//     normal_speed_task Outputs/csp_case_main_safety_air.sis.open_output.status <-> StandardOutputs/Air.csp_case_main_safety_air.sis.open_output.status_355
//     normal_speed_task Outputs/csp_case_main_safety_drives_PS2000.sis.open_output.status <-> StandardOutputs/DrivesRackPowerSupply.csp_case_main_safety_drives_PS2000.sis.open_output.status_57
//     normal_speed_task Outputs/csp_case_main_safety_drives_SD10000.sig.safety_group_err_ack_output.status <-> StandardOutputs/SD10000.ErrorAcknowledgement_35
//     normal_speed_task Outputs/csp_case_main_safety_drives_SD10100.sig.safety_group_err_ack_output.status <-> StandardOutputs/SD10100.ErrorAcknowledgement_37
//     normal_speed_task Outputs/csp_case_main_safety_drives_SD10200.sig.safety_group_err_ack_output.status <-> StandardOutputs/SD10200.ErrorAcknowledgement_39
//     normal_speed_task Outputs/csp_case_main_safety_drives_SD10300.sig.safety_group_err_ack_output.status <-> StandardOutputs/SD10300.ErrorAcknowledgement_41
//     normal_speed_task Outputs/csp_case_main_safety_drives_SD10400.sig.safety_group_err_ack_output.status <-> StandardOutputs/SD10400.ErrorAcknowledgement_43
//     normal_speed_task Outputs/csp_case_main_safety_drives_SD11000.sig.safety_group_err_ack_output.status <-> StandardOutputs/SD11000.ErrorAcknowledgement_45
//     normal_speed_task Outputs/csp_case_main_safety_drives_SD12000.sig.safety_group_err_ack_output.status <-> StandardOutputs/SD12000.ErrorAcknowledgement_19
//     normal_speed_task Outputs/csp_case_main_safety_drives_SD15000.sig.safety_group_err_ack_output.status <-> StandardOutputs/SD15000.ErrorAcknowledgement_47
//     normal_speed_task Outputs/csp_case_main_safety_drives_SD2100.sig.safety_group_err_ack_output.status <-> StandardOutputs/SD2100.ErrorAcknowledgement_9
//     normal_speed_task Outputs/csp_case_main_safety_drives_SD2200.sig.safety_group_err_ack_output.status <-> StandardOutputs/SD2200.ErrorAcknowledgement_11
//     normal_speed_task Outputs/csp_case_main_safety_drives_SD2300.sig.safety_group_err_ack_output.status <-> StandardOutputs/SD2300.ErrorAcknowledgement_13
//     normal_speed_task Outputs/csp_case_main_safety_drives_SD2400.sig.safety_group_err_ack_output.status <-> StandardOutputs/SD2400.ErrorAcknowledgement_15
//     normal_speed_task Outputs/csp_case_main_safety_drives_SD2500.sig.safety_group_err_ack_output.status <-> StandardOutputs/SD2500.ErrorAcknowledgement_17
//     normal_speed_task Outputs/csp_case_main_safety_drives_SD26000.sig.safety_group_err_ack_output.status <-> StandardOutputs/SD26000.ErrorAcknowledgement_49
//     normal_speed_task Outputs/csp_case_main_safety_drives_SD26100.sig.safety_group_err_ack_output.status <-> StandardOutputs/SD26100.ErrorAcknowledgement_51
//     normal_speed_task Outputs/csp_case_main_safety_drives_SD8000.sig.safety_group_err_ack_output.status <-> StandardOutputs/SD8000.ErrorAcknowledgement_21
//     normal_speed_task Outputs/csp_case_main_safety_drives_SD8100.sig.safety_group_err_ack_output.status <-> StandardOutputs/SD8100.ErrorAcknowledgement_23
//     normal_speed_task Outputs/csp_case_main_safety_drives_SD8200.sig.safety_group_err_ack_output.status <-> StandardOutputs/SD8200.ErrorAcknowledgement_25
//     normal_speed_task Outputs/csp_case_main_safety_drives_SD8300.sig.safety_group_err_ack_output.status <-> StandardOutputs/SD8300.ErrorAcknowledgement_27
//     normal_speed_task Outputs/csp_case_main_safety_drives_SD8400.sig.safety_group_err_ack_output.status <-> StandardOutputs/SD8400.ErrorAcknowledgement_29
//     normal_speed_task Outputs/csp_case_main_safety_drives_SD8500.sig.safety_group_err_ack_output.status <-> StandardOutputs/SD8500.ErrorAcknowledgement_31
//     normal_speed_task Outputs/csp_case_main_safety_drives_SD8600.sig.safety_group_err_ack_output.status <-> StandardOutputs/SD8600.ErrorAcknowledgement_33
//     normal_speed_task Outputs/csp_case_main_safety_drives_SD10000.sig.safety_group_run_output.status <-> StandardOutputs/SD10000.Run_36
//     normal_speed_task Outputs/csp_case_main_safety_drives_SD10100.sig.safety_group_run_output.status <-> StandardOutputs/SD10100.Run_38
//     normal_speed_task Outputs/csp_case_main_safety_drives_SD10200.sig.safety_group_run_output.status <-> StandardOutputs/SD10200.Run_40
//     normal_speed_task Outputs/csp_case_main_safety_drives_SD10300.sig.safety_group_run_output.status <-> StandardOutputs/SD10300.Run_42
//     normal_speed_task Outputs/csp_case_main_safety_drives_SD10400.sig.safety_group_run_output.status <-> StandardOutputs/SD10400.Run_44
//     normal_speed_task Outputs/csp_case_main_safety_drives_SD11000.sig.safety_group_run_output.status <-> StandardOutputs/SD11000.Run_46
//     normal_speed_task Outputs/csp_case_main_safety_drives_SD12000.sig.safety_group_run_output.status <-> StandardOutputs/SD12000.Run_20
//     normal_speed_task Outputs/csp_case_main_safety_drives_SD15000.sig.safety_group_run_output.status <-> StandardOutputs/SD15000.Run_48
//     normal_speed_task Outputs/csp_case_main_safety_drives_SD2100.sig.safety_group_run_output.status <-> StandardOutputs/SD2100.Run_10
//     normal_speed_task Outputs/csp_case_main_safety_drives_SD2200.sig.safety_group_run_output.status <-> StandardOutputs/SD2200.Run_12
//     normal_speed_task Outputs/csp_case_main_safety_drives_SD2300.sig.safety_group_run_output.status <-> StandardOutputs/SD2300.Run_14
//     normal_speed_task Outputs/csp_case_main_safety_drives_SD2400.sig.safety_group_run_output.status <-> StandardOutputs/SD2400.Run_16
//     normal_speed_task Outputs/csp_case_main_safety_drives_SD2500.sig.safety_group_run_output.status <-> StandardOutputs/SD2500.Run_18
//     normal_speed_task Outputs/csp_case_main_safety_drives_SD26000.sig.safety_group_run_output.status <-> StandardOutputs/SD26000.Run_50
//     normal_speed_task Outputs/csp_case_main_safety_drives_SD26100.sig.safety_group_run_output.status <-> StandardOutputs/SD26100.Run_52
//     normal_speed_task Outputs/csp_case_main_safety_drives_SD8000.sig.safety_group_run_output.status <-> StandardOutputs/SD8000.Run_22
//     normal_speed_task Outputs/csp_case_main_safety_drives_SD8100.sig.safety_group_run_output.status <-> StandardOutputs/SD8100.Run_24
//     normal_speed_task Outputs/csp_case_main_safety_drives_SD8200.sig.safety_group_run_output.status <-> StandardOutputs/SD8200.Run_26
//     normal_speed_task Outputs/csp_case_main_safety_drives_SD8300.sig.safety_group_run_output.status <-> StandardOutputs/SD8300.Run_28
//     normal_speed_task Outputs/csp_case_main_safety_drives_SD8400.sig.safety_group_run_output.status <-> StandardOutputs/SD8400.Run_30
//     normal_speed_task Outputs/csp_case_main_safety_drives_SD8500.sig.safety_group_run_output.status <-> StandardOutputs/SD8500.Run_32
//     normal_speed_task Outputs/csp_case_main_safety_drives_SD8600.sig.safety_group_run_output.status <-> StandardOutputs/SD8600.Run_34
//     normal_speed_task Outputs/csp_case_main_safety_emergency.sis.open_output.status <-> StandardOutputs/EmergencyCircuit.csp_case_main_safety_emergency.sis.open_output.status_65
//     normal_speed_task Outputs/csp_case_main_safety_guards.sis.open_output.status <-> StandardOutputs/Guards.csp_case_main_safety_guards.sis.open_output.status_274
//   SFI_CasePacker Instance <-> Cabinet ethercat master/CSPENC3/SPLC5000Slot14 (EL1819)
//     highest_speed_task Inputs/csp_case_feed_arm_sensors.case_feed_pb_di.field.status <-> Channel 12/Input
//     highest_speed_task Inputs/csp_case_glue_hotMelt.feeder_faulted_di.field.status <-> Channel 4/Input
//     highest_speed_task Inputs/csp_case_glue_hotMelt.level_ok_di.field.status <-> Channel 8/Input
//     highest_speed_task Inputs/csp_case_glue_hotMelt.ready_di.field.status <-> Channel 7/Input
//     low_speed_task Inputs/csp_case_main_safety_guards.sio_door_1.protection_safely_closed_input.status <-> Channel 1/Input
//     low_speed_task Inputs/csp_case_main_safety_guards.sio_door_2.protection_safely_closed_input.status <-> Channel 2/Input
//     low_speed_task Inputs/csp_main_jogManager.di_pendant_negative.field.status <-> Channel 12/Input
//     low_speed_task Inputs/csp_main_jogManager.di_pendant_positive.field.status <-> Channel 15/Input
//     lowest_speed_task Inputs/csp_case_main_cabinet.temperature_fault_di.field.status <-> Channel 3/Input
//   SFI_CasePacker Instance <-> Cabinet ethercat master/CSPENC3/SPLC5000Slot15 (EL1819)
//     highest_speed_task Inputs/csp_transfer_infeed_barcode_reader.Good_Read <-> Channel 7/Input
//     highest_speed_task Inputs/csp_transfer_infeed_barcode_reader.No_Read <-> Channel 8/Input
//     low_speed_task Inputs/csp_case_discharge_reject_modsort.modsort_fwd_faulted_di.field.status <-> Channel 1/Input
//     low_speed_task Inputs/csp_case_discharge_reject_modsort.modsort_reject_faulted_di.field.status <-> Channel 5/Input
//     lowest_speed_task Inputs/csp_case_main_cabinet.ups_alarm_di.field.status <-> Channel 3/Input
//     lowest_speed_task Inputs/csp_case_main_cabinet.ups_battery_charge_di.field.status <-> Channel 2/Input
//     lowest_speed_task Inputs/csp_case_main_cabinet.ups_battery_mode_di.field.status <-> Channel 6/Input
//   SFI_CasePacker Instance <-> Cabinet ethercat master/CSPENC3/SPLC5000Slot16 (EL2008)
//     highest_speed_task Outputs/csp_case_glue_hotMelt.standby_do.field.status <-> Channel 2/Output
//     normal_speed_task Outputs/csp_case_main_services.lights_on_do.field.status <-> Channel 8/Output
//     normal_speed_task Outputs/csp_case_main_services_airPressure.air_enable.field.status <-> Channel 7/Output
//     normal_speed_task Outputs/csp_case_main_services_pushbuttons.emergency_close_lamp_do.field.status <-> Channel 1/Output
//   SFI_CasePacker Instance <-> Cabinet ethercat master/CSPENC3/SPLC5000Slot17 (EL2008)
//     highest_speed_task Outputs/csp_case_discharge_reject_modsort.MODSORT_FWD_RUN_do.field.status <-> Channel 1/Output
//     highest_speed_task Outputs/csp_transfer_infeed_barcode_reader.Read_trigger <-> Channel 8/Output
//     highest_speed_task Outputs/csp_transfer_infeed_barcode_reader.teach_code_active <-> Channel 7/Output
//     normal_speed_task Outputs/csp_case_discharge_reject_modsort.MODSORT_REJECT_RUN_do.field.status <-> Channel 2/Output
//   SFI_CasePacker Instance <-> Cabinet ethercat master/CSPENC3/SPLC5000Slot18 (EL2008)
//     highest_speed_task Outputs/csp_transfer_infeed.temp_belt_run <-> Channel 1/Output
//   SFI_CasePacker Instance <-> Cabinet ethercat master/CSPENC3/SPLC5000Slot19 (EL6224)
//     highest_speed_task Inputs/csp_case_feed_arm_sensors.rfid_input_buffer.ByteArr[0] <-> IO-Link Port3_in/Bitheader 1
//     highest_speed_task Inputs/csp_case_feed_arm_sensors.rfid_input_buffer.ByteArr[9] <-> IO-Link Port3_in/Bitheader 2
//     highest_speed_task Inputs/csp_case_feed_arm_sensors.rfid_input_buffer.ByteArr[{1..8}] <-> IO-Link Port3_in/Byte {1..8}  (8 links)
//     highest_speed_task Inputs/csp_main_services.pressure_switch_value <-> IO-Link Port2/Pressure
//     highest_speed_task Outputs/csp_case_feed_arm_sensors.rfid_output_buffer.ByteArr[0] <-> IO-Link Port3_out/Bitheader 1
//     highest_speed_task Outputs/csp_case_feed_arm_sensors.rfid_output_buffer.ByteArr[9] <-> IO-Link Port3_out/Bitheader 2
//     highest_speed_task Outputs/csp_case_feed_arm_sensors.rfid_output_buffer.ByteArr[{1..8}] <-> IO-Link Port3_out/Byte {1..8}  (8 links)
//     normal_speed_task Inputs/csp_main_services.iol_master_el6224_IO6100.CONVERSION_private.process_data_input.AoeNetId <-> InfoData/AoeNetId
//     normal_speed_task Inputs/csp_main_services.iol_master_el6224_IO6100.CONVERSION_private.process_data_input.IOLinkDeviceStateInputs <-> DeviceState Inputs/State Ch1
//     normal_speed_task Inputs/csp_main_services.iol_master_el6224_IO6100.CONVERSION_private.process_data_input.IOLinkDeviceStateInputs @bit 8 <-> DeviceState Inputs/State Ch2
//     normal_speed_task Inputs/csp_main_services.iol_master_el6224_IO6100.CONVERSION_private.process_data_input.IOLinkDeviceStateInputs @bit 16 <-> DeviceState Inputs/State Ch3
//     normal_speed_task Inputs/csp_main_services.iol_master_el6224_IO6100.CONVERSION_private.process_data_input.IOLinkDeviceStateInputs @bit 24 <-> DeviceState Inputs/State Ch4
//     normal_speed_task Outputs/csp_main_services_towerLamp.buzzer_do.field.status <-> IO-Link Port1_out/Buzzer State
//     normal_speed_task Outputs/csp_main_services_towerLamp.buzzer_volume <-> IO-Link Port1_out/Buzzer Volume
//     normal_speed_task Outputs/csp_main_services_towerLamp.tower_lamp.iol_slave_pdo_output.blinking_freq <-> IO-Link Port1_out/Blinking frequency / Level value high byte / Running speed
//     normal_speed_task Outputs/csp_main_services_towerLamp.tower_lamp.iol_slave_pdo_output.number_segments <-> IO-Link Port1_out/Number of segments / Level type
//     normal_speed_task Outputs/csp_main_services_towerLamp.tower_lamp.iol_slave_pdo_output.operating_mode <-> IO-Link Port1_out/Operating mode
//     normal_speed_task Outputs/csp_main_services_towerLamp.tower_lamp.iol_slave_pdo_output.seg_1_blink <-> IO-Link Port1_out/Segment 1 blink / dominant / LED4
//     normal_speed_task Outputs/csp_main_services_towerLamp.tower_lamp.iol_slave_pdo_output.seg_2_blink <-> IO-Link Port1_out/Segment 2 blink / dominant / LED8
//     normal_speed_task Outputs/csp_main_services_towerLamp.tower_lamp.iol_slave_pdo_output.seg_3_blink <-> IO-Link Port1_out/Segment 3 blink / dominant / LED12
//     normal_speed_task Outputs/csp_main_services_towerLamp.tower_lamp.iol_slave_pdo_output.seg_1_color <-> IO-Link Port1_out/Segment 1 color / Background color / LED3-1
//     normal_speed_task Outputs/csp_main_services_towerLamp.tower_lamp.iol_slave_pdo_output.seg_2_color <-> IO-Link Port1_out/Segment 2 color / Running color / LED7-5
//     normal_speed_task Outputs/csp_main_services_towerLamp.tower_lamp.iol_slave_pdo_output.seg_3_color <-> IO-Link Port1_out/Segment 3 color / LED11-9
//   SFI_CasePacker Instance <-> Cabinet ethercat master/CSPENC3/SPLC5000Slot20 (EL4004)
//     normal_speed_task Outputs/csp_case_discharge_reject.modsort_belt_speed_analog_reference_ao.field.value <-> AO Outputs Channel 1/Analog output
//   SFI_CasePacker Instance <-> Cabinet ethercat master/CSPENC3/SPLC5000Slot21(EK1122-0008)/Box 92 (EP2328-0001)
//     highest_speed_task Outputs/csp_case_glue.os_lower_gun_1_do.field.status <-> Channel 7/Output
//     highest_speed_task Outputs/csp_case_glue.os_lower_gun_2_do.field.status <-> Channel 8/Output
//     highest_speed_task Outputs/csp_case_glue.os_upper_gun_1_do.field.status <-> Channel 5/Output
//     highest_speed_task Outputs/csp_case_glue.os_upper_gun_2_do.field.status <-> Channel 6/Output
//   SFI_CasePacker Instance <-> Cabinet ethercat master/CSPENC3/SPLC5000Slot21(EK1122-0008)/Box 93 (EP2328-0001)
//     highest_speed_task Outputs/csp_case_glue.ls_lower_gun_1_do.field.status <-> Channel 7/Output
//     highest_speed_task Outputs/csp_case_glue.ls_lower_gun_2_do.field.status <-> Channel 8/Output
//     highest_speed_task Outputs/csp_case_glue.ls_upper_gun_1_do.field.status <-> Channel 5/Output
//     highest_speed_task Outputs/csp_case_glue.ls_upper_gun_2_do.field.status <-> Channel 6/Output
//   SFI_CasePacker Instance <-> Cabinet ethercat master/CSPENC3/SPLC5000Slot21(EK1122-0008)/IOB11120 (EP1018-0001)
//     highest_speed_task Inputs/csp_case_fc_ls_upper_sensors.flap_di.field.status <-> Channel 3/Input
//     highest_speed_task Inputs/csp_case_glue_sensors.case_present_ls_di.field.status <-> Channel 4/Input
//     normal_speed_task Inputs/csp_case_openFlap_sensors.open_flap_ls_di.field.status <-> Channel 2/Input
//   SFI_CasePacker Instance <-> Cabinet ethercat master/CSPENC3/SPLC5000Slot21(EK1122-0008)/IOB11130 (EP1018-0001)
//     highest_speed_task Inputs/csp_case_fc_os_upper_sensors.flap_di.field.status <-> Channel 3/Input
//     highest_speed_task Inputs/csp_case_glue_sensors.case_present_os_di.field.status <-> Channel 4/Input
//     normal_speed_task Inputs/csp_case_openFlap_sensors.open_flap_os_di.field.status <-> Channel 2/Input
//   SFI_CasePacker Instance <-> Cabinet ethercat master/CSPENC3/SPLC5000Slot21(EK1122-0008)/IOB15120 (EP1018-0001)
//     low_speed_task Inputs/csp_case_discharge_reject_sensors.downstream_backup_di.field.status <-> Channel 2/Input
//     low_speed_task Inputs/csp_case_discharge_reject_sensors.reject_backup_di.field.status <-> Channel 3/Input
//     low_speed_task Inputs/csp_case_discharge_reject_sensors.reject_present_di.field.status <-> Channel 4/Input
//     normal_speed_task Inputs/csp_case_discharge_reject_sensors.reject_trigger_di.field.status <-> Channel 1/Input
//   SFI_CasePacker Instance <-> Cabinet ethercat master/CSPENC3/SPLC5000Slot21(EK1122-0008)/IOB8800 (EP2318-0001)
//     highest_speed_task Inputs/csp_case_feed_arm_sensors.case_check_di.field.status <-> Channel 1/Input
//     highest_speed_task Outputs/csp_case_feed_arm_sensors.major_vacuum_do.field.status <-> Channel 5/Output
//     highest_speed_task Outputs/csp_case_feed_arm_sensors.minor_vacuum_do.field.status <-> Channel 7/Output
//     low_speed_task Outputs/csp_case_tr_accU_virtualMaster.brake_release_do.field.status <-> Channel 6/Output
//   SFI_CasePacker Instance <-> Cabinet ethercat master/HMI6600 (CPXXXX-BK1150)
//     normal_speed_task Inputs/csp_case_main_services_pushbuttons.reset_di.field.status <-> Term 2 (CPx9xx-8)/Channel 1/Key 1
//     normal_speed_task Inputs/csp_case_main_services_pushbuttons.start_di.field.status <-> Term 2 (CPx9xx-8)/Channel 1/Key 3
//     normal_speed_task Inputs/csp_case_main_services_pushbuttons.stop_di.field.status <-> Term 2 (CPx9xx-8)/Channel 1/Key 2
//     normal_speed_task Outputs/csp_case_main_services_pushbuttons.reset_lamp_do.field.status <-> Term 2 (CPx9xx-8)/Channel 1/LED 1
//     normal_speed_task Outputs/csp_case_main_services_pushbuttons.start_lamp_do.field.status <-> Term 2 (CPx9xx-8)/Channel 1/LED 3
//     normal_speed_task Outputs/csp_case_main_services_pushbuttons.stop_lamp_do.field.status <-> Term 2 (CPx9xx-8)/Channel 1/LED 2
//   SFI_CasePacker Instance <-> Cabinet ethercat master/IO61000 (EK1100)/IO6100Slot24 (EL7211)
//     low_speed_task Inputs/csp_case_transport_accU_depth.Slot24_drv.process_data_input.status_word <-> DRV Statusword/Statusword
//     low_speed_task Inputs/csp_case_transport_accU_depth.axis.hard_increments.value <-> FB Position/Position
//     lowest_speed_task Inputs/csp_case_transport_accU_depth.NC_encoder_val <-> FB Position/Position
//   SFI_CasePacker Instance <-> Cabinet ethercat master/IO61000 (EK1100)/IO6100Slot26 (EL7211)
//     low_speed_task Inputs/csp_case_feed_shuttle_accU_depth.Slot26_drv.process_data_input.status_word <-> DRV Statusword/Statusword
//     low_speed_task Inputs/csp_case_feed_shuttle_accU_depth.axis.hard_increments.value <-> FB Position/Position
//     lowest_speed_task Inputs/csp_case_feed_shuttle_accU_depth.NC_encoder_val <-> FB Position/Position
//   SFI_CasePacker Instance <-> Cabinet ethercat master/IO61000 (EK1100)/IO6100Slot29 (EL7211)
//     low_speed_task Inputs/csp_case_feed_magazine_accU_lsDepth.Slot29_drv.process_data_input.status_word <-> DRV Statusword/Statusword
//     low_speed_task Inputs/csp_case_feed_magazine_accU_lsDepth.axis.hard_increments.value <-> FB Position/Position
//     lowest_speed_task Inputs/csp_case_feed_magazine_accU_lsDepth.NC_encoder_val <-> FB Position/Position
//   SFI_CasePacker Instance <-> Cabinet ethercat master/IO61000 (EK1100)/IO6100Slot31 (EL7211)
//     low_speed_task Inputs/csp_case_feed_magazine_accU_osDepth.Slot31_drv.process_data_input.status_word <-> DRV Statusword/Statusword
//     low_speed_task Inputs/csp_case_feed_magazine_accU_osDepth.axis.hard_increments.value <-> FB Position/Position
//     lowest_speed_task Inputs/csp_case_feed_magazine_accU_osDepth.NC_encoder_val <-> FB Position/Position
//   SFI_CasePacker Instance <-> Cabinet ethercat master/IO61000 (EK1100)/IO6100Slot34 (EL7221)
//     low_speed_task Inputs/csp_case_loader_guide_accU_width.Slot34_drv.process_data_input.status_word <-> DRV Statusword/Statusword
//     low_speed_task Inputs/csp_case_loader_guide_accU_width.axis.hard_increments.value <-> FB Position/Position
//     lowest_speed_task Inputs/csp_case_loader_guide_accU_width.NC_encoder_val <-> FB Position/Position
//   SFI_CasePacker Instance <-> Cabinet ethercat master/IO61000 (EK1100)/IO6100Slot36 (EL7211)
//     low_speed_task Inputs/csp_case_glue_os_accU_width.Slot36_drv.process_data_input.status_word <-> DRV Statusword/Statusword
//     low_speed_task Inputs/csp_case_glue_os_accU_width.axis.hard_increments.value <-> FB Position/Position
//     lowest_speed_task Inputs/csp_case_glue_os_accU_width.NC_encoder_val <-> FB Position/Position
//   SFI_CasePacker Instance <-> Cabinet ethercat master/IO61000 (EK1100)/IO6100Slot39 (EL7211)
//     low_speed_task Inputs/csp_case_glue_os_accU_upperPosition.Slot39_drv.process_data_input.status_word <-> DRV Statusword/Statusword
//     low_speed_task Inputs/csp_case_glue_os_accU_upperPosition.axis.hard_increments.value <-> FB Position/Position
//     lowest_speed_task Inputs/csp_case_glue_os_accU_upperPosition.NC_encoder_val <-> FB Position/Position
//   SFI_CasePacker Instance <-> Cabinet ethercat master/IO61000 (EK1100)/IO6100Slot41 (EL7211)
//     low_speed_task Inputs/csp_case_glue_os_accU_lowerPosition.Slot41_drv.process_data_input.status_word <-> DRV Statusword/Statusword
//     low_speed_task Inputs/csp_case_glue_os_accU_lowerPosition.axis.hard_increments.value <-> FB Position/Position
//     lowest_speed_task Inputs/csp_case_glue_os_accU_lowerPosition.NC_encoder_val <-> FB Position/Position
//   SFI_CasePacker Instance <-> Cabinet ethercat master/IO61000 (EK1100)/IO6100Slot44 (EL7211)
//     low_speed_task Inputs/csp_case_glue_ls_accU_upperPosition.Slot44_drv.process_data_input.status_word <-> DRV Statusword/Statusword
//     low_speed_task Inputs/csp_case_glue_ls_accU_upperPosition.axis.hard_increments.value <-> FB Position/Position
//     lowest_speed_task Inputs/csp_case_glue_ls_accU_upperPosition.NC_encoder_val <-> FB Position/Position
//   SFI_CasePacker Instance <-> Cabinet ethercat master/IO61000 (EK1100)/IO6100Slot46 (EL7211)
//     low_speed_task Inputs/csp_case_glue_ls_accU_lowerPosition.Slot46_drv.process_data_input.status_word <-> DRV Statusword/Statusword
//     low_speed_task Inputs/csp_case_glue_ls_accU_lowerPosition.axis.hard_increments.value <-> FB Position/Position
//     lowest_speed_task Inputs/csp_case_glue_ls_accU_lowerPosition.NC_encoder_val <-> FB Position/Position
//   SFI_CasePacker Instance <-> Cabinet ethercat master/IO61000 (EK1100)/IO6100Slot49 (EL7211)
//     low_speed_task Inputs/csp_case_feed_reject_accU_depth.Slot49_drv.process_data_input.status_word <-> DRV Statusword/Statusword
//     low_speed_task Inputs/csp_case_feed_reject_accU_depth.axis.hard_increments.value <-> FB Position/Position
//     lowest_speed_task Inputs/csp_case_feed_reject_accU_depth.NC_encoder_val <-> FB Position/Position
//   SFI_CasePacker Instance <-> Cabinet ethercat master/IO61000 (EK1100)/IO6100Slot51 (EL7211)
//     low_speed_task Inputs/csp_case_tr_accU_os_width.Slot51_drv.process_data_input.status_word <-> DRV Statusword/Statusword
//     low_speed_task Inputs/csp_case_tr_accU_os_width.axis.hard_increments.value <-> FB Position/Position
//     lowest_speed_task Inputs/csp_case_tr_accU_os_width.NC_encoder_val <-> FB Position/Position
//   SFI_CasePacker Instance <-> Cabinet ethercat master/IO61000 (EK1100)/IO6100Slot55 (EL7211)
//     low_speed_task Inputs/csp_case_tr_accU_ls_width.Slot55_drv.process_data_input.status_word <-> DRV Statusword/Statusword
//     low_speed_task Inputs/csp_case_tr_accU_ls_width.axis.hard_increments.value <-> FB Position/Position
//     lowest_speed_task Inputs/csp_case_tr_accU_ls_width.NC_encoder_val <-> FB Position/Position
//   SFI_CasePacker Instance <-> Cabinet ethercat master/IO61000 (EK1100)/IO6100Slot57 (EL7211)
//     low_speed_task Inputs/csp_case_tr_accU_depth.Slot57_drv.process_data_input.status_word <-> DRV Statusword/Statusword
//     low_speed_task Inputs/csp_case_tr_accU_depth.axis.hard_increments.value <-> FB Position/Position
//     lowest_speed_task Inputs/csp_case_tr_accU_depth.NC_encoder_val <-> FB Position/Position
//   SFI_CasePacker Instance <-> Cabinet ethercat master/IOB2820 (EP2318-0001)
//     highest_speed_task Inputs/csp_case_fc_ls_lower_sensors.flap_di.field.status <-> Channel 1/Input
//     normal_speed_task Inputs/csp_case_openFlap_sensors.open_trailing_minor_di.field.status <-> Channel 3/Input
//   SFI_CasePacker Instance <-> Cabinet ethercat master/IOB2830 (EP2318-0001)
//     highest_speed_task Inputs/csp_case_fc_os_lower_sensors.flap_di.field.status <-> Channel 2/Input
//     low_speed_task Inputs/csp_case_transport_os_minorPlow.bwd_di.field.status <-> Channel 4/Input
//     low_speed_task Inputs/csp_case_transport_os_minorPlow.fwd_di.field.status <-> Channel 3/Input
//     normal_speed_task Inputs/csp_case_flapControl_backStop.present_di.field.status <-> Channel 1/Input
//     normal_speed_task Outputs/csp_case_flapControl_backStop.extend_do.field.status <-> Channel 5/Output
//     normal_speed_task Outputs/csp_case_transport_tensioner.chain_tensioner_do.field.status <-> Channel 7/Output
//   SFI_CasePacker Instance <-> Cabinet ethercat master/IOB3020 (EP6224-2022)
//     highest_speed_task Inputs/csp_case_closing.ls_rfid_input_buffer.ByteArr[0] <-> IO-Link Port3_in/Bitheader 1
//     highest_speed_task Inputs/csp_case_closing.ls_rfid_input_buffer.ByteArr[9] <-> IO-Link Port3_in/Bitheader 2
//     highest_speed_task Inputs/csp_case_closing.ls_rfid_input_buffer.ByteArr[{1..8}] <-> IO-Link Port3_in/Byte {1..8}  (8 links)
//     highest_speed_task Outputs/csp_case_closing.ls_rfid_output_buffer.ByteArr[0] <-> IO-Link Port3_out/Bitheader 1
//     highest_speed_task Outputs/csp_case_closing.ls_rfid_output_buffer.ByteArr[9] <-> IO-Link Port3_out/Bitheader 2
//     highest_speed_task Outputs/csp_case_closing.ls_rfid_output_buffer.ByteArr[{1..8}] <-> IO-Link Port3_out/Byte {1..8}  (8 links)
//     normal_speed_task Inputs/csp_case_loader_sensors.rfid_input_buffer.ByteArr[0] <-> IO-Link Port2_in/Bitheader 1
//     normal_speed_task Inputs/csp_case_loader_sensors.rfid_input_buffer.ByteArr[9] <-> IO-Link Port2_in/Bitheader 2
//     normal_speed_task Inputs/csp_case_loader_sensors.rfid_input_buffer.ByteArr[{1..8}] <-> IO-Link Port2_in/Byte {1..8}  (8 links)
//     normal_speed_task Outputs/csp_case_loader_sensors.rfid_output_buffer.ByteArr[0] <-> IO-Link Port2_out/Bitheader 1
//     normal_speed_task Outputs/csp_case_loader_sensors.rfid_output_buffer.ByteArr[9] <-> IO-Link Port2_out/Bitheader 2
//     normal_speed_task Outputs/csp_case_loader_sensors.rfid_output_buffer.ByteArr[{1..8}] <-> IO-Link Port2_out/Byte {1..8}  (8 links)
//   SFI_CasePacker Instance <-> Cabinet ethercat master/IOB3030 (EP6224-2022)
//     highest_speed_task Inputs/csp_case_closing.os_rfid_input_buffer.ByteArr[0] <-> IO-Link Port3_in/Bitheader 1
//     highest_speed_task Inputs/csp_case_closing.os_rfid_input_buffer.ByteArr[9] <-> IO-Link Port3_in/Bitheader 2
//     highest_speed_task Inputs/csp_case_closing.os_rfid_input_buffer.ByteArr[{1..8}] <-> IO-Link Port3_in/Byte {1..8}  (8 links)
//     highest_speed_task Outputs/csp_case_closing.os_rfid_output_buffer.ByteArr[0] <-> IO-Link Port3_out/Bitheader 1
//     highest_speed_task Outputs/csp_case_closing.os_rfid_output_buffer.ByteArr[9] <-> IO-Link Port3_out/Bitheader 2
//     highest_speed_task Outputs/csp_case_closing.os_rfid_output_buffer.ByteArr[{1..8}] <-> IO-Link Port3_out/Byte {1..8}  (8 links)
//   SFI_CasePacker Instance <-> Cabinet ethercat master/IOB8810 (EP2008-0001)
//     low_speed_task Outputs/csp_case_feed_magazine_ls_pusher.retract_do.field.status <-> Channel 2/Output
//     low_speed_task Outputs/csp_case_feed_magazine_ls_pusherTilt.extend_do.field.status <-> Channel 4/Output
//     low_speed_task Outputs/csp_case_feed_magazine_os_pusher.retract_do.field.status <-> Channel 1/Output
//     low_speed_task Outputs/csp_case_feed_magazine_os_pusherTilt.extend_do.field.status <-> Channel 3/Output
//   SFI_CasePacker Instance <-> Cabinet ethercat master/IOB8820 (EP1018-0001)
//     low_speed_task Inputs/csp_case_feed_magazine_level_zone4.di.field.status <-> Channel 1/Input
//     normal_speed_task Inputs/csp_case_feed_magazine_level_zone2.di.field.status <-> Channel 3/Input
//     normal_speed_task Inputs/csp_case_feed_magazine_level_zone3.di.field.status <-> Channel 2/Input
//     normal_speed_task Inputs/csp_case_feed_magazine_ls_pusher.retracted_di.field.status <-> Channel 6/Input
//     normal_speed_task Inputs/csp_case_feed_magazine_ls_pusherTilt.upstream_di.field.status <-> Channel 7/Input
//   SFI_CasePacker Instance <-> Cabinet ethercat master/IOB8830 (EP1018-0001)
//     low_speed_task Inputs/csp_case_feed_magazine_ls_pusherTilt.downstream_di.field.status <-> Channel 6/Input
//     low_speed_task Inputs/csp_case_feed_magazine_ls_sensors.feed_di.field.status <-> Channel 2/Input
//     normal_speed_task Inputs/csp_case_feed_magazine_level_zone1.di.field.status <-> Channel 4/Input
//     normal_speed_task Inputs/csp_case_feed_magazine_level_zonelow.di.field.status <-> Channel 5/Input
//     normal_speed_task Inputs/csp_case_feed_magazine_level_zonemin.di.field.status <-> Channel 3/Input
//   SFI_CasePacker Instance <-> Cabinet ethercat master/IOB8900 (EP1018-0001)
//     low_speed_task Inputs/csp_case_feed_magazine_os_pusherTilt.downstream_di.field.status <-> Channel 4/Input
//     low_speed_task Inputs/csp_case_feed_magazine_os_sensors.feed_di.field.status <-> Channel 3/Input
//     normal_speed_task Inputs/csp_case_feed_magazine_os_pusher.retracted_di.field.status <-> Channel 1/Input
//     normal_speed_task Inputs/csp_case_feed_magazine_os_pusherTilt.upstream_di.field.status <-> Channel 2/Input
//   SFI_CasePacker Instance <-> Cabinet ethercat master/MAN8920 (CPX-FB37)
//     highest_speed_task Outputs/csp_case_feed_shuttle_sensors.vacuum1_do.field.status <-> Module 3 (VTSA DIL 4 [32DO])/Outputs/Output 0
//     highest_speed_task Outputs/csp_case_feed_shuttle_sensors.vacuum2_do.field.status <-> Module 3 (VTSA DIL 4 [32DO])/Outputs/Output 1
//     highest_speed_task Outputs/csp_case_feed_shuttle_sensors.vacuum3_do.field.status <-> Module 3 (VTSA DIL 4 [32DO])/Outputs/Output 3
//     highest_speed_task Outputs/csp_case_feed_shuttle_sensors.vacuum4_do.field.status <-> Module 3 (VTSA DIL 4 [32DO])/Outputs/Output 2
//     highest_speed_task Outputs/csp_case_feed_shuttle_sensors.vacuum5_do.field.status <-> Module 3 (VTSA DIL 4 [32DO])/Outputs/Output 4
//     highest_speed_task Outputs/csp_case_feed_shuttle_sensors.vacuum6_do.field.status <-> Module 3 (VTSA DIL 4 [32DO])/Outputs/Output 5
//     highest_speed_task Outputs/csp_case_feed_shuttle_sensors.vacuum7_do.field.status <-> Module 3 (VTSA DIL 4 [32DO])/Outputs/Output 6
//   SFI_CasePacker Instance <-> Cabinet ethercat master/SD10000
//     highest_speed_task Inputs/csp_case_main_drives.SD10000_drv.channel_a.process_data_input.dc_bus_power <-> AT 1/DC bus power
//     highest_speed_task Inputs/csp_case_main_drives.SD10000_drv.channel_a.process_data_input.dc_bus_voltage <-> AT 1/DC bus voltage
//     highest_speed_task Inputs/csp_case_main_drives.SD10000_drv.channel_a.process_data_input.motor_temperature <-> AT 1/Motor temperature
//     highest_speed_task Inputs/csp_case_main_drives.SD10000_drv.channel_b.process_data_input.dc_bus_power <-> AT 2/DC bus power
//     highest_speed_task Inputs/csp_case_main_drives.SD10000_drv.channel_b.process_data_input.dc_bus_voltage <-> AT 2/DC bus voltage
//     highest_speed_task Inputs/csp_case_main_drives.SD10000_drv.channel_b.process_data_input.motor_temperature <-> AT 2/Motor temperature
//     normal_speed_task Inputs/csp_case_main_drives.SD10000_drv.channel_a.process_data_input.actual_absolute_current <-> AT 1/Torque-generating current, actual value
//     normal_speed_task Inputs/csp_case_main_drives.SD10000_drv.channel_a.process_data_input.dc_bus_ready <-> AT 1/Device control: Status word[15]
//     normal_speed_task Inputs/csp_case_main_drives.SD10000_drv.channel_a.process_data_input.status_parametrization_level <-> AT 1/Status parametrization level
//     normal_speed_task Inputs/csp_case_main_drives.SD10000_drv.channel_a.process_data_input.warning_active <-> AT 1/Device control: Status word[2]
//     normal_speed_task Inputs/csp_case_main_drives.SD10000_drv.channel_b.process_data_input.actual_absolute_current <-> AT 2/Torque-generating current, actual value
//     normal_speed_task Inputs/csp_case_main_drives.SD10000_drv.channel_b.process_data_input.dc_bus_ready <-> AT 2/Device control: Status word[15]
//     normal_speed_task Inputs/csp_case_main_drives.SD10000_drv.channel_b.process_data_input.status_parametrization_level <-> AT 2/Status parametrization level
//     normal_speed_task Inputs/csp_case_main_drives.SD10000_drv.channel_b.process_data_input.warning_active <-> AT 2/Device control: Status word[2]
//   SFI_CasePacker Instance <-> Cabinet ethercat master/SD10100
//     highest_speed_task Inputs/csp_case_main_drives.SD10100_drv.channel_a.process_data_input.dc_bus_power <-> AT 1/DC bus power
//     highest_speed_task Inputs/csp_case_main_drives.SD10100_drv.channel_a.process_data_input.dc_bus_voltage <-> AT 1/DC bus voltage
//     highest_speed_task Inputs/csp_case_main_drives.SD10100_drv.channel_a.process_data_input.motor_temperature <-> AT 1/Motor temperature
//     highest_speed_task Inputs/csp_case_main_drives.SD10100_drv.channel_b.process_data_input.dc_bus_power <-> AT 2/DC bus power
//     highest_speed_task Inputs/csp_case_main_drives.SD10100_drv.channel_b.process_data_input.dc_bus_voltage <-> AT 2/DC bus voltage
//     highest_speed_task Inputs/csp_case_main_drives.SD10100_drv.channel_b.process_data_input.motor_temperature <-> AT 2/Motor temperature
//     normal_speed_task Inputs/csp_case_main_drives.SD10100_drv.channel_a.process_data_input.actual_absolute_current <-> AT 1/Torque-generating current, actual value
//     normal_speed_task Inputs/csp_case_main_drives.SD10100_drv.channel_a.process_data_input.dc_bus_ready <-> AT 1/Device control: Status word[15]
//     normal_speed_task Inputs/csp_case_main_drives.SD10100_drv.channel_a.process_data_input.status_parametrization_level <-> AT 1/Status parametrization level
//     normal_speed_task Inputs/csp_case_main_drives.SD10100_drv.channel_a.process_data_input.warning_active <-> AT 1/Device control: Status word[2]
//     normal_speed_task Inputs/csp_case_main_drives.SD10100_drv.channel_b.process_data_input.actual_absolute_current <-> AT 2/Torque-generating current, actual value
//     normal_speed_task Inputs/csp_case_main_drives.SD10100_drv.channel_b.process_data_input.dc_bus_ready <-> AT 2/Device control: Status word[15]
//     normal_speed_task Inputs/csp_case_main_drives.SD10100_drv.channel_b.process_data_input.status_parametrization_level <-> AT 2/Status parametrization level
//     normal_speed_task Inputs/csp_case_main_drives.SD10100_drv.channel_b.process_data_input.warning_active <-> AT 2/Device control: Status word[2]
//   SFI_CasePacker Instance <-> Cabinet ethercat master/SD10200
//     highest_speed_task Inputs/csp_case_main_drives.SD10200_drv.channel_a.process_data_input.dc_bus_power <-> AT 1/DC bus power
//     highest_speed_task Inputs/csp_case_main_drives.SD10200_drv.channel_a.process_data_input.dc_bus_voltage <-> AT 1/DC bus voltage
//     highest_speed_task Inputs/csp_case_main_drives.SD10200_drv.channel_a.process_data_input.motor_temperature <-> AT 1/Motor temperature
//     highest_speed_task Inputs/csp_case_main_drives.SD10200_drv.channel_b.process_data_input.dc_bus_power <-> AT 2/DC bus power
//     highest_speed_task Inputs/csp_case_main_drives.SD10200_drv.channel_b.process_data_input.dc_bus_voltage <-> AT 2/DC bus voltage
//     highest_speed_task Inputs/csp_case_main_drives.SD10200_drv.channel_b.process_data_input.motor_temperature <-> AT 2/Motor temperature
//     normal_speed_task Inputs/csp_case_main_drives.SD10200_drv.channel_a.process_data_input.actual_absolute_current <-> AT 1/Torque-generating current, actual value
//     normal_speed_task Inputs/csp_case_main_drives.SD10200_drv.channel_a.process_data_input.dc_bus_ready <-> AT 1/Device control: Status word[15]
//     normal_speed_task Inputs/csp_case_main_drives.SD10200_drv.channel_a.process_data_input.status_parametrization_level <-> AT 1/Status parametrization level
//     normal_speed_task Inputs/csp_case_main_drives.SD10200_drv.channel_a.process_data_input.warning_active <-> AT 1/Device control: Status word[2]
//     normal_speed_task Inputs/csp_case_main_drives.SD10200_drv.channel_b.process_data_input.actual_absolute_current <-> AT 2/Torque-generating current, actual value
//     normal_speed_task Inputs/csp_case_main_drives.SD10200_drv.channel_b.process_data_input.dc_bus_ready <-> AT 2/Device control: Status word[15]
//     normal_speed_task Inputs/csp_case_main_drives.SD10200_drv.channel_b.process_data_input.status_parametrization_level <-> AT 2/Status parametrization level
//     normal_speed_task Inputs/csp_case_main_drives.SD10200_drv.channel_b.process_data_input.warning_active <-> AT 2/Device control: Status word[2]
//   SFI_CasePacker Instance <-> Cabinet ethercat master/SD10300
//     highest_speed_task Inputs/csp_case_main_drives.SD10300_drv.channel_a.process_data_input.dc_bus_power <-> AT 1/DC bus power
//     highest_speed_task Inputs/csp_case_main_drives.SD10300_drv.channel_a.process_data_input.dc_bus_voltage <-> AT 1/DC bus voltage
//     highest_speed_task Inputs/csp_case_main_drives.SD10300_drv.channel_a.process_data_input.motor_temperature <-> AT 1/Motor temperature
//     highest_speed_task Inputs/csp_case_main_drives.SD10300_drv.channel_b.process_data_input.dc_bus_power <-> AT 2/DC bus power
//     highest_speed_task Inputs/csp_case_main_drives.SD10300_drv.channel_b.process_data_input.dc_bus_voltage <-> AT 2/DC bus voltage
//     highest_speed_task Inputs/csp_case_main_drives.SD10300_drv.channel_b.process_data_input.motor_temperature <-> AT 2/Motor temperature
//     normal_speed_task Inputs/csp_case_main_drives.SD10300_drv.channel_a.process_data_input.actual_absolute_current <-> AT 1/Torque-generating current, actual value
//     normal_speed_task Inputs/csp_case_main_drives.SD10300_drv.channel_a.process_data_input.dc_bus_ready <-> AT 1/Device control: Status word[15]
//     normal_speed_task Inputs/csp_case_main_drives.SD10300_drv.channel_a.process_data_input.status_parametrization_level <-> AT 1/Status parametrization level
//     normal_speed_task Inputs/csp_case_main_drives.SD10300_drv.channel_a.process_data_input.warning_active <-> AT 1/Device control: Status word[2]
//     normal_speed_task Inputs/csp_case_main_drives.SD10300_drv.channel_b.process_data_input.actual_absolute_current <-> AT 2/Torque-generating current, actual value
//     normal_speed_task Inputs/csp_case_main_drives.SD10300_drv.channel_b.process_data_input.dc_bus_ready <-> AT 2/Device control: Status word[15]
//     normal_speed_task Inputs/csp_case_main_drives.SD10300_drv.channel_b.process_data_input.status_parametrization_level <-> AT 2/Status parametrization level
//     normal_speed_task Inputs/csp_case_main_drives.SD10300_drv.channel_b.process_data_input.warning_active <-> AT 2/Device control: Status word[2]
//   SFI_CasePacker Instance <-> Cabinet ethercat master/SD10400
//     highest_speed_task Inputs/csp_case_main_drives.SD10400_drv.channel_a.process_data_input.dc_bus_power <-> AT 1/DC bus power
//     highest_speed_task Inputs/csp_case_main_drives.SD10400_drv.channel_a.process_data_input.dc_bus_voltage <-> AT 1/DC bus voltage
//     highest_speed_task Inputs/csp_case_main_drives.SD10400_drv.channel_a.process_data_input.motor_temperature <-> AT 1/Motor temperature
//     highest_speed_task Inputs/csp_case_main_drives.SD10400_drv.channel_b.process_data_input.dc_bus_power <-> AT 2/DC bus power
//     highest_speed_task Inputs/csp_case_main_drives.SD10400_drv.channel_b.process_data_input.dc_bus_voltage <-> AT 2/DC bus voltage
//     highest_speed_task Inputs/csp_case_main_drives.SD10400_drv.channel_b.process_data_input.motor_temperature <-> AT 2/Motor temperature
//     normal_speed_task Inputs/csp_case_main_drives.SD10400_drv.channel_a.process_data_input.actual_absolute_current <-> AT 1/Torque-generating current, actual value
//     normal_speed_task Inputs/csp_case_main_drives.SD10400_drv.channel_a.process_data_input.dc_bus_ready <-> AT 1/Device control: Status word[15]
//     normal_speed_task Inputs/csp_case_main_drives.SD10400_drv.channel_a.process_data_input.status_parametrization_level <-> AT 1/Status parametrization level
//     normal_speed_task Inputs/csp_case_main_drives.SD10400_drv.channel_a.process_data_input.warning_active <-> AT 1/Device control: Status word[2]
//     normal_speed_task Inputs/csp_case_main_drives.SD10400_drv.channel_b.process_data_input.actual_absolute_current <-> AT 2/Torque-generating current, actual value
//     normal_speed_task Inputs/csp_case_main_drives.SD10400_drv.channel_b.process_data_input.dc_bus_ready <-> AT 2/Device control: Status word[15]
//     normal_speed_task Inputs/csp_case_main_drives.SD10400_drv.channel_b.process_data_input.status_parametrization_level <-> AT 2/Status parametrization level
//     normal_speed_task Inputs/csp_case_main_drives.SD10400_drv.channel_b.process_data_input.warning_active <-> AT 2/Device control: Status word[2]
//   SFI_CasePacker Instance <-> Cabinet ethercat master/SD11000
//     normal_speed_task Inputs/csp_case_main_drives.SD11000_drv.channel_a.process_data_input.actual_absolute_current <-> AT 1/Torque-generating current, actual value
//     normal_speed_task Inputs/csp_case_main_drives.SD11000_drv.channel_a.process_data_input.dc_bus_power <-> AT 1/DC bus power
//     normal_speed_task Inputs/csp_case_main_drives.SD11000_drv.channel_a.process_data_input.dc_bus_ready <-> AT 1/Device control: Status word[15]
//     normal_speed_task Inputs/csp_case_main_drives.SD11000_drv.channel_a.process_data_input.dc_bus_voltage <-> AT 1/DC bus voltage
//     normal_speed_task Inputs/csp_case_main_drives.SD11000_drv.channel_a.process_data_input.motor_temperature <-> AT 1/Motor temperature
//     normal_speed_task Inputs/csp_case_main_drives.SD11000_drv.channel_a.process_data_input.status_parametrization_level <-> AT 1/Status parametrization level
//     normal_speed_task Inputs/csp_case_main_drives.SD11000_drv.channel_a.process_data_input.warning_active <-> AT 1/Device control: Status word[2]
//   SFI_CasePacker Instance <-> Cabinet ethercat master/SD12000
//     normal_speed_task Inputs/csp_case_main_drives.SD12000_drv.channel_a.process_data_input.actual_absolute_current <-> AT 1/Torque-generating current, actual value
//     normal_speed_task Inputs/csp_case_main_drives.SD12000_drv.channel_a.process_data_input.dc_bus_power <-> AT 1/DC bus power
//     normal_speed_task Inputs/csp_case_main_drives.SD12000_drv.channel_a.process_data_input.dc_bus_ready <-> AT 1/Device control: Status word[15]
//     normal_speed_task Inputs/csp_case_main_drives.SD12000_drv.channel_a.process_data_input.dc_bus_voltage <-> AT 1/DC bus voltage
//     normal_speed_task Inputs/csp_case_main_drives.SD12000_drv.channel_a.process_data_input.motor_temperature <-> AT 1/Motor temperature
//     normal_speed_task Inputs/csp_case_main_drives.SD12000_drv.channel_a.process_data_input.status_parametrization_level <-> AT 1/Status parametrization level
//     normal_speed_task Inputs/csp_case_main_drives.SD12000_drv.channel_a.process_data_input.warning_active <-> AT 1/Device control: Status word[2]
//     normal_speed_task Inputs/csp_case_main_drives.SD12000_drv.channel_b.process_data_input.actual_absolute_current <-> AT 2/Torque-generating current, actual value
//     normal_speed_task Inputs/csp_case_main_drives.SD12000_drv.channel_b.process_data_input.dc_bus_power <-> AT 2/DC bus power
//     normal_speed_task Inputs/csp_case_main_drives.SD12000_drv.channel_b.process_data_input.dc_bus_ready <-> AT 2/Device control: Status word[15]
//     normal_speed_task Inputs/csp_case_main_drives.SD12000_drv.channel_b.process_data_input.dc_bus_voltage <-> AT 2/DC bus voltage
//     normal_speed_task Inputs/csp_case_main_drives.SD12000_drv.channel_b.process_data_input.motor_temperature <-> AT 2/Motor temperature
//     normal_speed_task Inputs/csp_case_main_drives.SD12000_drv.channel_b.process_data_input.status_parametrization_level <-> AT 2/Status parametrization level
//     normal_speed_task Inputs/csp_case_main_drives.SD12000_drv.channel_b.process_data_input.warning_active <-> AT 2/Device control: Status word[2]
//   SFI_CasePacker Instance <-> Cabinet ethercat master/SD2100
//     highest_speed_task Inputs/csp_case_main_drives.SD2100_drv.channel_a.process_data_input.dc_bus_power <-> AT 1/DC bus power
//     highest_speed_task Inputs/csp_case_main_drives.SD2100_drv.channel_a.process_data_input.dc_bus_voltage <-> AT 1/DC bus voltage
//     highest_speed_task Inputs/csp_case_main_drives.SD2100_drv.channel_a.process_data_input.motor_temperature <-> AT 1/Motor temperature
//     highest_speed_task Inputs/csp_case_main_drives.SD2100_drv.channel_b.process_data_input.dc_bus_power <-> AT 2/DC bus power
//     highest_speed_task Inputs/csp_case_main_drives.SD2100_drv.channel_b.process_data_input.dc_bus_voltage <-> AT 2/DC bus voltage
//     highest_speed_task Inputs/csp_case_main_drives.SD2100_drv.channel_b.process_data_input.motor_temperature <-> AT 2/Motor temperature
//     normal_speed_task Inputs/csp_case_main_drives.SD2100_drv.channel_a.process_data_input.actual_absolute_current <-> AT 1/Torque-generating current, actual value
//     normal_speed_task Inputs/csp_case_main_drives.SD2100_drv.channel_a.process_data_input.dc_bus_ready <-> AT 1/Device control: Status word[15]
//     normal_speed_task Inputs/csp_case_main_drives.SD2100_drv.channel_a.process_data_input.status_parametrization_level <-> AT 1/Status parametrization level
//     normal_speed_task Inputs/csp_case_main_drives.SD2100_drv.channel_a.process_data_input.warning_active <-> AT 1/Device control: Status word[2]
//     normal_speed_task Inputs/csp_case_main_drives.SD2100_drv.channel_b.process_data_input.actual_absolute_current <-> AT 2/Torque-generating current, actual value
//     normal_speed_task Inputs/csp_case_main_drives.SD2100_drv.channel_b.process_data_input.dc_bus_ready <-> AT 2/Device control: Status word[15]
//     normal_speed_task Inputs/csp_case_main_drives.SD2100_drv.channel_b.process_data_input.status_parametrization_level <-> AT 2/Status parametrization level
//     normal_speed_task Inputs/csp_case_main_drives.SD2100_drv.channel_b.process_data_input.warning_active <-> AT 2/Device control: Status word[2]
//   SFI_CasePacker Instance <-> Cabinet ethercat master/SD2200
//     highest_speed_task Inputs/csp_case_main_drives.SD2200_drv.channel_a.process_data_input.dc_bus_power <-> AT 1/DC bus power
//     highest_speed_task Inputs/csp_case_main_drives.SD2200_drv.channel_a.process_data_input.dc_bus_voltage <-> AT 1/DC bus voltage
//     highest_speed_task Inputs/csp_case_main_drives.SD2200_drv.channel_a.process_data_input.motor_temperature <-> AT 1/Motor temperature
//     highest_speed_task Inputs/csp_case_main_drives.SD2200_drv.channel_b.process_data_input.dc_bus_power <-> AT 2/DC bus power
//     highest_speed_task Inputs/csp_case_main_drives.SD2200_drv.channel_b.process_data_input.dc_bus_voltage <-> AT 2/DC bus voltage
//     highest_speed_task Inputs/csp_case_main_drives.SD2200_drv.channel_b.process_data_input.motor_temperature <-> AT 2/Motor temperature
//     normal_speed_task Inputs/csp_case_main_drives.SD2200_drv.channel_a.process_data_input.actual_absolute_current <-> AT 1/Torque-generating current, actual value
//     normal_speed_task Inputs/csp_case_main_drives.SD2200_drv.channel_a.process_data_input.dc_bus_ready <-> AT 1/Device control: Status word[15]
//     normal_speed_task Inputs/csp_case_main_drives.SD2200_drv.channel_a.process_data_input.status_parametrization_level <-> AT 1/Status parametrization level
//     normal_speed_task Inputs/csp_case_main_drives.SD2200_drv.channel_a.process_data_input.warning_active <-> AT 1/Device control: Status word[2]
//     normal_speed_task Inputs/csp_case_main_drives.SD2200_drv.channel_b.process_data_input.actual_absolute_current <-> AT 2/Torque-generating current, actual value
//     normal_speed_task Inputs/csp_case_main_drives.SD2200_drv.channel_b.process_data_input.dc_bus_ready <-> AT 2/Device control: Status word[15]
//     normal_speed_task Inputs/csp_case_main_drives.SD2200_drv.channel_b.process_data_input.status_parametrization_level <-> AT 2/Status parametrization level
//     normal_speed_task Inputs/csp_case_main_drives.SD2200_drv.channel_b.process_data_input.warning_active <-> AT 2/Device control: Status word[2]
//   SFI_CasePacker Instance <-> Cabinet ethercat master/SD2300
//     highest_speed_task Inputs/csp_case_main_drives.SD2300_drv.channel_a.process_data_input.dc_bus_power <-> AT 1/DC bus power
//     highest_speed_task Inputs/csp_case_main_drives.SD2300_drv.channel_a.process_data_input.dc_bus_voltage <-> AT 1/DC bus voltage
//     highest_speed_task Inputs/csp_case_main_drives.SD2300_drv.channel_a.process_data_input.motor_temperature <-> AT 1/Motor temperature
//     highest_speed_task Inputs/csp_case_main_drives.SD2300_drv.channel_b.process_data_input.dc_bus_power <-> AT 2/DC bus power
//     highest_speed_task Inputs/csp_case_main_drives.SD2300_drv.channel_b.process_data_input.dc_bus_voltage <-> AT 2/DC bus voltage
//     highest_speed_task Inputs/csp_case_main_drives.SD2300_drv.channel_b.process_data_input.motor_temperature <-> AT 2/Motor temperature
//     normal_speed_task Inputs/csp_case_main_drives.SD2300_drv.channel_a.process_data_input.actual_absolute_current <-> AT 1/Torque-generating current, actual value
//     normal_speed_task Inputs/csp_case_main_drives.SD2300_drv.channel_a.process_data_input.dc_bus_ready <-> AT 1/Device control: Status word[15]
//     normal_speed_task Inputs/csp_case_main_drives.SD2300_drv.channel_a.process_data_input.status_parametrization_level <-> AT 1/Status parametrization level
//     normal_speed_task Inputs/csp_case_main_drives.SD2300_drv.channel_a.process_data_input.warning_active <-> AT 1/Device control: Status word[2]
//     normal_speed_task Inputs/csp_case_main_drives.SD2300_drv.channel_b.process_data_input.actual_absolute_current <-> AT 2/Torque-generating current, actual value
//     normal_speed_task Inputs/csp_case_main_drives.SD2300_drv.channel_b.process_data_input.dc_bus_ready <-> AT 2/Device control: Status word[15]
//     normal_speed_task Inputs/csp_case_main_drives.SD2300_drv.channel_b.process_data_input.status_parametrization_level <-> AT 2/Status parametrization level
//     normal_speed_task Inputs/csp_case_main_drives.SD2300_drv.channel_b.process_data_input.warning_active <-> AT 2/Device control: Status word[2]
//   SFI_CasePacker Instance <-> Cabinet ethercat master/SD2400
//     highest_speed_task Inputs/csp_case_main_drives.SD2400_drv.channel_a.process_data_input.dc_bus_power <-> AT 1/DC bus power
//     highest_speed_task Inputs/csp_case_main_drives.SD2400_drv.channel_a.process_data_input.dc_bus_voltage <-> AT 1/DC bus voltage
//     highest_speed_task Inputs/csp_case_main_drives.SD2400_drv.channel_a.process_data_input.motor_temperature <-> AT 1/Motor temperature
//     highest_speed_task Inputs/csp_case_main_drives.SD2400_drv.channel_b.process_data_input.dc_bus_power <-> AT 2/DC bus power
//     highest_speed_task Inputs/csp_case_main_drives.SD2400_drv.channel_b.process_data_input.dc_bus_voltage <-> AT 2/DC bus voltage
//     highest_speed_task Inputs/csp_case_main_drives.SD2400_drv.channel_b.process_data_input.motor_temperature <-> AT 2/Motor temperature
//     normal_speed_task Inputs/csp_case_main_drives.SD2400_drv.channel_a.process_data_input.actual_absolute_current <-> AT 1/Torque-generating current, actual value
//     normal_speed_task Inputs/csp_case_main_drives.SD2400_drv.channel_a.process_data_input.dc_bus_ready <-> AT 1/Device control: Status word[15]
//     normal_speed_task Inputs/csp_case_main_drives.SD2400_drv.channel_a.process_data_input.status_parametrization_level <-> AT 1/Status parametrization level
//     normal_speed_task Inputs/csp_case_main_drives.SD2400_drv.channel_a.process_data_input.warning_active <-> AT 1/Device control: Status word[2]
//     normal_speed_task Inputs/csp_case_main_drives.SD2400_drv.channel_b.process_data_input.actual_absolute_current <-> AT 2/Torque-generating current, actual value
//     normal_speed_task Inputs/csp_case_main_drives.SD2400_drv.channel_b.process_data_input.dc_bus_ready <-> AT 2/Device control: Status word[15]
//     normal_speed_task Inputs/csp_case_main_drives.SD2400_drv.channel_b.process_data_input.status_parametrization_level <-> AT 2/Status parametrization level
//     normal_speed_task Inputs/csp_case_main_drives.SD2400_drv.channel_b.process_data_input.warning_active <-> AT 2/Device control: Status word[2]
//   SFI_CasePacker Instance <-> Cabinet ethercat master/SD2500
//     highest_speed_task Inputs/csp_case_main_drives.SD2500_drv.channel_a.process_data_input.dc_bus_power <-> AT 1/DC bus power
//     highest_speed_task Inputs/csp_case_main_drives.SD2500_drv.channel_a.process_data_input.dc_bus_voltage <-> AT 1/DC bus voltage
//     highest_speed_task Inputs/csp_case_main_drives.SD2500_drv.channel_a.process_data_input.motor_temperature <-> AT 1/Motor temperature
//     highest_speed_task Inputs/csp_case_main_drives.SD2500_drv.channel_b.process_data_input.dc_bus_power <-> AT 2/DC bus power
//     highest_speed_task Inputs/csp_case_main_drives.SD2500_drv.channel_b.process_data_input.dc_bus_voltage <-> AT 2/DC bus voltage
//     highest_speed_task Inputs/csp_case_main_drives.SD2500_drv.channel_b.process_data_input.motor_temperature <-> AT 2/Motor temperature
//     normal_speed_task Inputs/csp_case_main_drives.SD2500_drv.channel_a.process_data_input.actual_absolute_current <-> AT 1/Torque-generating current, actual value
//     normal_speed_task Inputs/csp_case_main_drives.SD2500_drv.channel_a.process_data_input.dc_bus_ready <-> AT 1/Device control: Status word[15]
//     normal_speed_task Inputs/csp_case_main_drives.SD2500_drv.channel_a.process_data_input.status_parametrization_level <-> AT 1/Status parametrization level
//     normal_speed_task Inputs/csp_case_main_drives.SD2500_drv.channel_a.process_data_input.warning_active <-> AT 1/Device control: Status word[2]
//     normal_speed_task Inputs/csp_case_main_drives.SD2500_drv.channel_b.process_data_input.actual_absolute_current <-> AT 2/Torque-generating current, actual value
//     normal_speed_task Inputs/csp_case_main_drives.SD2500_drv.channel_b.process_data_input.dc_bus_ready <-> AT 2/Device control: Status word[15]
//     normal_speed_task Inputs/csp_case_main_drives.SD2500_drv.channel_b.process_data_input.status_parametrization_level <-> AT 2/Status parametrization level
//     normal_speed_task Inputs/csp_case_main_drives.SD2500_drv.channel_b.process_data_input.warning_active <-> AT 2/Device control: Status word[2]
//   SFI_CasePacker Instance <-> Cabinet ethercat master/SD26000
//     normal_speed_task Inputs/csp_case_main_drives.SD26000_drv.channel_a.process_data_input.actual_absolute_current <-> AT 1/Torque-generating current, actual value
//     normal_speed_task Inputs/csp_case_main_drives.SD26000_drv.channel_a.process_data_input.dc_bus_power <-> AT 1/DC bus power
//     normal_speed_task Inputs/csp_case_main_drives.SD26000_drv.channel_a.process_data_input.dc_bus_ready <-> AT 1/Device control: Status word[15]
//     normal_speed_task Inputs/csp_case_main_drives.SD26000_drv.channel_a.process_data_input.dc_bus_voltage <-> AT 1/DC bus voltage
//     normal_speed_task Inputs/csp_case_main_drives.SD26000_drv.channel_a.process_data_input.motor_temperature <-> AT 1/Motor temperature
//     normal_speed_task Inputs/csp_case_main_drives.SD26000_drv.channel_a.process_data_input.status_parametrization_level <-> AT 1/Status parametrization level
//     normal_speed_task Inputs/csp_case_main_drives.SD26000_drv.channel_a.process_data_input.warning_active <-> AT 1/Device control: Status word[2]
//     normal_speed_task Inputs/csp_case_main_drives.SD26000_drv.channel_b.process_data_input.actual_absolute_current <-> AT 2/Torque-generating current, actual value
//     normal_speed_task Inputs/csp_case_main_drives.SD26000_drv.channel_b.process_data_input.dc_bus_power <-> AT 2/DC bus power
//     normal_speed_task Inputs/csp_case_main_drives.SD26000_drv.channel_b.process_data_input.dc_bus_ready <-> AT 2/Device control: Status word[15]
//     normal_speed_task Inputs/csp_case_main_drives.SD26000_drv.channel_b.process_data_input.dc_bus_voltage <-> AT 2/DC bus voltage
//     normal_speed_task Inputs/csp_case_main_drives.SD26000_drv.channel_b.process_data_input.motor_temperature <-> AT 2/Motor temperature
//     normal_speed_task Inputs/csp_case_main_drives.SD26000_drv.channel_b.process_data_input.status_parametrization_level <-> AT 2/Status parametrization level
//     normal_speed_task Inputs/csp_case_main_drives.SD26000_drv.channel_b.process_data_input.warning_active <-> AT 2/Device control: Status word[2]
//   SFI_CasePacker Instance <-> Cabinet ethercat master/SD26100
//     normal_speed_task Inputs/csp_case_main_drives.SD26100_drv.channel_a.process_data_input.actual_absolute_current <-> AT 1/Torque-generating current, actual value
//     normal_speed_task Inputs/csp_case_main_drives.SD26100_drv.channel_a.process_data_input.dc_bus_power <-> AT 1/DC bus power
//     normal_speed_task Inputs/csp_case_main_drives.SD26100_drv.channel_a.process_data_input.dc_bus_ready <-> AT 1/Device control: Status word[15]
//     normal_speed_task Inputs/csp_case_main_drives.SD26100_drv.channel_a.process_data_input.dc_bus_voltage <-> AT 1/DC bus voltage
//     normal_speed_task Inputs/csp_case_main_drives.SD26100_drv.channel_a.process_data_input.motor_temperature <-> AT 1/Motor temperature
//     normal_speed_task Inputs/csp_case_main_drives.SD26100_drv.channel_a.process_data_input.status_parametrization_level <-> AT 1/Status parametrization level
//     normal_speed_task Inputs/csp_case_main_drives.SD26100_drv.channel_a.process_data_input.warning_active <-> AT 1/Device control: Status word[2]
//     normal_speed_task Inputs/csp_case_main_drives.SD26100_drv.channel_b.process_data_input.actual_absolute_current <-> AT 2/Torque-generating current, actual value
//     normal_speed_task Inputs/csp_case_main_drives.SD26100_drv.channel_b.process_data_input.dc_bus_power <-> AT 2/DC bus power
//     normal_speed_task Inputs/csp_case_main_drives.SD26100_drv.channel_b.process_data_input.dc_bus_ready <-> AT 2/Device control: Status word[15]
//     normal_speed_task Inputs/csp_case_main_drives.SD26100_drv.channel_b.process_data_input.dc_bus_voltage <-> AT 2/DC bus voltage
//     normal_speed_task Inputs/csp_case_main_drives.SD26100_drv.channel_b.process_data_input.motor_temperature <-> AT 2/Motor temperature
//     normal_speed_task Inputs/csp_case_main_drives.SD26100_drv.channel_b.process_data_input.status_parametrization_level <-> AT 2/Status parametrization level
//     normal_speed_task Inputs/csp_case_main_drives.SD26100_drv.channel_b.process_data_input.warning_active <-> AT 2/Device control: Status word[2]
//   SFI_CasePacker Instance <-> Cabinet ethercat master/SD8000
//     highest_speed_task Inputs/csp_case_main_drives.SD8000_drv.channel_a.process_data_input.dc_bus_power <-> AT 1/DC bus power
//     highest_speed_task Inputs/csp_case_main_drives.SD8000_drv.channel_a.process_data_input.dc_bus_voltage <-> AT 1/DC bus voltage
//     highest_speed_task Inputs/csp_case_main_drives.SD8000_drv.channel_a.process_data_input.motor_temperature <-> AT 1/Motor temperature
//     highest_speed_task Inputs/csp_case_main_drives.SD8000_drv.channel_b.process_data_input.dc_bus_power <-> AT 2/DC bus power
//     highest_speed_task Inputs/csp_case_main_drives.SD8000_drv.channel_b.process_data_input.dc_bus_voltage <-> AT 2/DC bus voltage
//     highest_speed_task Inputs/csp_case_main_drives.SD8000_drv.channel_b.process_data_input.motor_temperature <-> AT 2/Motor temperature
//     normal_speed_task Inputs/csp_case_main_drives.SD8000_drv.channel_a.process_data_input.actual_absolute_current <-> AT 1/Torque-generating current, actual value
//     normal_speed_task Inputs/csp_case_main_drives.SD8000_drv.channel_a.process_data_input.dc_bus_ready <-> AT 1/Device control: Status word[15]
//     normal_speed_task Inputs/csp_case_main_drives.SD8000_drv.channel_a.process_data_input.status_parametrization_level <-> AT 1/Status parametrization level
//     normal_speed_task Inputs/csp_case_main_drives.SD8000_drv.channel_a.process_data_input.warning_active <-> AT 1/Device control: Status word[2]
//     normal_speed_task Inputs/csp_case_main_drives.SD8000_drv.channel_b.process_data_input.actual_absolute_current <-> AT 2/Torque-generating current, actual value
//     normal_speed_task Inputs/csp_case_main_drives.SD8000_drv.channel_b.process_data_input.dc_bus_ready <-> AT 2/Device control: Status word[15]
//     normal_speed_task Inputs/csp_case_main_drives.SD8000_drv.channel_b.process_data_input.status_parametrization_level <-> AT 2/Status parametrization level
//     normal_speed_task Inputs/csp_case_main_drives.SD8000_drv.channel_b.process_data_input.warning_active <-> AT 2/Device control: Status word[2]
//   SFI_CasePacker Instance <-> Cabinet ethercat master/SD8100
//     highest_speed_task Inputs/csp_case_main_drives.SD8100_drv.channel_a.process_data_input.dc_bus_power <-> AT 1/DC bus power
//     highest_speed_task Inputs/csp_case_main_drives.SD8100_drv.channel_a.process_data_input.dc_bus_voltage <-> AT 1/DC bus voltage
//     highest_speed_task Inputs/csp_case_main_drives.SD8100_drv.channel_a.process_data_input.motor_temperature <-> AT 1/Motor temperature
//     highest_speed_task Inputs/csp_case_main_drives.SD8100_drv.channel_b.process_data_input.dc_bus_power <-> AT 2/DC bus power
//     highest_speed_task Inputs/csp_case_main_drives.SD8100_drv.channel_b.process_data_input.dc_bus_voltage <-> AT 2/DC bus voltage
//     highest_speed_task Inputs/csp_case_main_drives.SD8100_drv.channel_b.process_data_input.motor_temperature <-> AT 2/Motor temperature
//     normal_speed_task Inputs/csp_case_main_drives.SD8100_drv.channel_a.process_data_input.actual_absolute_current <-> AT 1/Torque-generating current, actual value
//     normal_speed_task Inputs/csp_case_main_drives.SD8100_drv.channel_a.process_data_input.dc_bus_ready <-> AT 1/Device control: Status word[15]
//     normal_speed_task Inputs/csp_case_main_drives.SD8100_drv.channel_a.process_data_input.status_parametrization_level <-> AT 1/Status parametrization level
//     normal_speed_task Inputs/csp_case_main_drives.SD8100_drv.channel_a.process_data_input.warning_active <-> AT 1/Device control: Status word[2]
//     normal_speed_task Inputs/csp_case_main_drives.SD8100_drv.channel_b.process_data_input.actual_absolute_current <-> AT 2/Torque-generating current, actual value
//     normal_speed_task Inputs/csp_case_main_drives.SD8100_drv.channel_b.process_data_input.dc_bus_ready <-> AT 2/Device control: Status word[15]
//     normal_speed_task Inputs/csp_case_main_drives.SD8100_drv.channel_b.process_data_input.status_parametrization_level <-> AT 2/Status parametrization level
//     normal_speed_task Inputs/csp_case_main_drives.SD8100_drv.channel_b.process_data_input.warning_active <-> AT 2/Device control: Status word[2]
//   SFI_CasePacker Instance <-> Cabinet ethercat master/SD8200
//     highest_speed_task Inputs/csp_case_main_drives.SD8200_drv.channel_a.process_data_input.dc_bus_power <-> AT 1/DC bus power
//     highest_speed_task Inputs/csp_case_main_drives.SD8200_drv.channel_a.process_data_input.dc_bus_voltage <-> AT 1/DC bus voltage
//     highest_speed_task Inputs/csp_case_main_drives.SD8200_drv.channel_a.process_data_input.motor_temperature <-> AT 1/Motor temperature
//     highest_speed_task Inputs/csp_case_main_drives.SD8200_drv.channel_b.process_data_input.dc_bus_power <-> AT 2/DC bus power
//     highest_speed_task Inputs/csp_case_main_drives.SD8200_drv.channel_b.process_data_input.dc_bus_voltage <-> AT 2/DC bus voltage
//     highest_speed_task Inputs/csp_case_main_drives.SD8200_drv.channel_b.process_data_input.motor_temperature <-> AT 2/Motor temperature
//     normal_speed_task Inputs/csp_case_main_drives.SD8200_drv.channel_a.process_data_input.actual_absolute_current <-> AT 1/Torque-generating current, actual value
//     normal_speed_task Inputs/csp_case_main_drives.SD8200_drv.channel_a.process_data_input.dc_bus_ready <-> AT 1/Device control: Status word[15]
//     normal_speed_task Inputs/csp_case_main_drives.SD8200_drv.channel_a.process_data_input.status_parametrization_level <-> AT 1/Status parametrization level
//     normal_speed_task Inputs/csp_case_main_drives.SD8200_drv.channel_a.process_data_input.warning_active <-> AT 1/Device control: Status word[2]
//     normal_speed_task Inputs/csp_case_main_drives.SD8200_drv.channel_b.process_data_input.actual_absolute_current <-> AT 2/Torque-generating current, actual value
//     normal_speed_task Inputs/csp_case_main_drives.SD8200_drv.channel_b.process_data_input.dc_bus_ready <-> AT 2/Device control: Status word[15]
//     normal_speed_task Inputs/csp_case_main_drives.SD8200_drv.channel_b.process_data_input.status_parametrization_level <-> AT 2/Status parametrization level
//     normal_speed_task Inputs/csp_case_main_drives.SD8200_drv.channel_b.process_data_input.warning_active <-> AT 2/Device control: Status word[2]
//   SFI_CasePacker Instance <-> Cabinet ethercat master/SD8300
//     highest_speed_task Inputs/csp_case_main_drives.SD8300_drv.channel_a.process_data_input.dc_bus_power <-> AT 1/DC bus power
//     highest_speed_task Inputs/csp_case_main_drives.SD8300_drv.channel_a.process_data_input.dc_bus_voltage <-> AT 1/DC bus voltage
//     highest_speed_task Inputs/csp_case_main_drives.SD8300_drv.channel_a.process_data_input.motor_temperature <-> AT 1/Motor temperature
//     highest_speed_task Inputs/csp_case_main_drives.SD8300_drv.channel_b.process_data_input.dc_bus_power <-> AT 2/DC bus power
//     highest_speed_task Inputs/csp_case_main_drives.SD8300_drv.channel_b.process_data_input.dc_bus_voltage <-> AT 2/DC bus voltage
//     highest_speed_task Inputs/csp_case_main_drives.SD8300_drv.channel_b.process_data_input.motor_temperature <-> AT 2/Motor temperature
//     normal_speed_task Inputs/csp_case_main_drives.SD8300_drv.channel_a.process_data_input.actual_absolute_current <-> AT 1/Torque-generating current, actual value
//     normal_speed_task Inputs/csp_case_main_drives.SD8300_drv.channel_a.process_data_input.dc_bus_ready <-> AT 1/Device control: Status word[15]
//     normal_speed_task Inputs/csp_case_main_drives.SD8300_drv.channel_a.process_data_input.status_parametrization_level <-> AT 1/Status parametrization level
//     normal_speed_task Inputs/csp_case_main_drives.SD8300_drv.channel_a.process_data_input.warning_active <-> AT 1/Device control: Status word[2]
//     normal_speed_task Inputs/csp_case_main_drives.SD8300_drv.channel_b.process_data_input.actual_absolute_current <-> AT 2/Torque-generating current, actual value
//     normal_speed_task Inputs/csp_case_main_drives.SD8300_drv.channel_b.process_data_input.dc_bus_ready <-> AT 2/Device control: Status word[15]
//     normal_speed_task Inputs/csp_case_main_drives.SD8300_drv.channel_b.process_data_input.status_parametrization_level <-> AT 2/Status parametrization level
//     normal_speed_task Inputs/csp_case_main_drives.SD8300_drv.channel_b.process_data_input.warning_active <-> AT 2/Device control: Status word[2]
//   SFI_CasePacker Instance <-> Cabinet ethercat master/SD8400
//     normal_speed_task Inputs/csp_case_main_drives.SD8400_drv.channel_a.process_data_input.actual_absolute_current <-> AT 1/Torque-generating current, actual value
//     normal_speed_task Inputs/csp_case_main_drives.SD8400_drv.channel_a.process_data_input.dc_bus_power <-> AT 1/DC bus power
//     normal_speed_task Inputs/csp_case_main_drives.SD8400_drv.channel_a.process_data_input.dc_bus_ready <-> AT 1/Device control: Status word[15]
//     normal_speed_task Inputs/csp_case_main_drives.SD8400_drv.channel_a.process_data_input.dc_bus_voltage <-> AT 1/DC bus voltage
//     normal_speed_task Inputs/csp_case_main_drives.SD8400_drv.channel_a.process_data_input.motor_temperature <-> AT 1/Motor temperature
//     normal_speed_task Inputs/csp_case_main_drives.SD8400_drv.channel_a.process_data_input.status_parametrization_level <-> AT 1/Status parametrization level
//     normal_speed_task Inputs/csp_case_main_drives.SD8400_drv.channel_a.process_data_input.warning_active <-> AT 1/Device control: Status word[2]
//     normal_speed_task Inputs/csp_case_main_drives.SD8400_drv.channel_b.process_data_input.actual_absolute_current <-> AT 2/Torque-generating current, actual value
//     normal_speed_task Inputs/csp_case_main_drives.SD8400_drv.channel_b.process_data_input.dc_bus_power <-> AT 2/DC bus power
//     normal_speed_task Inputs/csp_case_main_drives.SD8400_drv.channel_b.process_data_input.dc_bus_ready <-> AT 2/Device control: Status word[15]
//     normal_speed_task Inputs/csp_case_main_drives.SD8400_drv.channel_b.process_data_input.dc_bus_voltage <-> AT 2/DC bus voltage
//     normal_speed_task Inputs/csp_case_main_drives.SD8400_drv.channel_b.process_data_input.motor_temperature <-> AT 2/Motor temperature
//     normal_speed_task Inputs/csp_case_main_drives.SD8400_drv.channel_b.process_data_input.status_parametrization_level <-> AT 2/Status parametrization level
//     normal_speed_task Inputs/csp_case_main_drives.SD8400_drv.channel_b.process_data_input.warning_active <-> AT 2/Device control: Status word[2]
//   SFI_CasePacker Instance <-> Cabinet ethercat master/SD8500
//     highest_speed_task Inputs/csp_case_main_drives.SD8500_drv.channel_a.process_data_input.dc_bus_power <-> AT 1/DC bus power
//     highest_speed_task Inputs/csp_case_main_drives.SD8500_drv.channel_a.process_data_input.dc_bus_voltage <-> AT 1/DC bus voltage
//     highest_speed_task Inputs/csp_case_main_drives.SD8500_drv.channel_a.process_data_input.motor_temperature <-> AT 1/Motor temperature
//     highest_speed_task Inputs/csp_case_main_drives.SD8500_drv.channel_b.process_data_input.dc_bus_power <-> AT 2/DC bus power
//     highest_speed_task Inputs/csp_case_main_drives.SD8500_drv.channel_b.process_data_input.dc_bus_voltage <-> AT 2/DC bus voltage
//     highest_speed_task Inputs/csp_case_main_drives.SD8500_drv.channel_b.process_data_input.motor_temperature <-> AT 2/Motor temperature
//     normal_speed_task Inputs/csp_case_main_drives.SD8500_drv.channel_a.process_data_input.actual_absolute_current <-> AT 1/Torque-generating current, actual value
//     normal_speed_task Inputs/csp_case_main_drives.SD8500_drv.channel_a.process_data_input.dc_bus_ready <-> AT 1/Device control: Status word[15]
//     normal_speed_task Inputs/csp_case_main_drives.SD8500_drv.channel_a.process_data_input.status_parametrization_level <-> AT 1/Status parametrization level
//     normal_speed_task Inputs/csp_case_main_drives.SD8500_drv.channel_a.process_data_input.warning_active <-> AT 1/Device control: Status word[2]
//     normal_speed_task Inputs/csp_case_main_drives.SD8500_drv.channel_b.process_data_input.actual_absolute_current <-> AT 2/Torque-generating current, actual value
//     normal_speed_task Inputs/csp_case_main_drives.SD8500_drv.channel_b.process_data_input.dc_bus_ready <-> AT 2/Device control: Status word[15]
//     normal_speed_task Inputs/csp_case_main_drives.SD8500_drv.channel_b.process_data_input.status_parametrization_level <-> AT 2/Status parametrization level
//     normal_speed_task Inputs/csp_case_main_drives.SD8500_drv.channel_b.process_data_input.warning_active <-> AT 2/Device control: Status word[2]
//   SFI_CasePacker Instance <-> Cabinet ethercat master/SD8600
//     normal_speed_task Inputs/csp_case_main_drives.SD8600_drv.channel_a.process_data_input.actual_absolute_current <-> AT 1/Torque-generating current, actual value
//     normal_speed_task Inputs/csp_case_main_drives.SD8600_drv.channel_a.process_data_input.dc_bus_power <-> AT 1/DC bus power
//     normal_speed_task Inputs/csp_case_main_drives.SD8600_drv.channel_a.process_data_input.dc_bus_ready <-> AT 1/Device control: Status word[15]
//     normal_speed_task Inputs/csp_case_main_drives.SD8600_drv.channel_a.process_data_input.dc_bus_voltage <-> AT 1/DC bus voltage
//     normal_speed_task Inputs/csp_case_main_drives.SD8600_drv.channel_a.process_data_input.motor_temperature <-> AT 1/Motor temperature
//     normal_speed_task Inputs/csp_case_main_drives.SD8600_drv.channel_a.process_data_input.status_parametrization_level <-> AT 1/Status parametrization level
//     normal_speed_task Inputs/csp_case_main_drives.SD8600_drv.channel_a.process_data_input.warning_active <-> AT 1/Device control: Status word[2]
//     normal_speed_task Inputs/csp_case_main_drives.SD8600_drv.channel_b.process_data_input.actual_absolute_current <-> AT 2/Torque-generating current, actual value
//     normal_speed_task Inputs/csp_case_main_drives.SD8600_drv.channel_b.process_data_input.dc_bus_power <-> AT 2/DC bus power
//     normal_speed_task Inputs/csp_case_main_drives.SD8600_drv.channel_b.process_data_input.dc_bus_ready <-> AT 2/Device control: Status word[15]
//     normal_speed_task Inputs/csp_case_main_drives.SD8600_drv.channel_b.process_data_input.dc_bus_voltage <-> AT 2/DC bus voltage
//     normal_speed_task Inputs/csp_case_main_drives.SD8600_drv.channel_b.process_data_input.motor_temperature <-> AT 2/Motor temperature
//     normal_speed_task Inputs/csp_case_main_drives.SD8600_drv.channel_b.process_data_input.status_parametrization_level <-> AT 2/Status parametrization level
//     normal_speed_task Inputs/csp_case_main_drives.SD8600_drv.channel_b.process_data_input.warning_active <-> AT 2/Device control: Status word[2]
//   SFI_CasePacker Instance <-> Device 2 (EtherCAT Automation Protocol, EL6601)/Box 95 (Publisher)
//     normal_speed_task Outputs/.RAJ_to_Flexlink <-> RAJ_To_FLexlink_Var/Outputs/VarData
//   SFI_CasePacker Instance <-> Device 2 (EtherCAT Automation Protocol, EL6601)/Box 96 (Subscriber)
//     normal_speed_task Inputs/.Flexlink_to_RAJ <-> Flexlink_To_RAJ_Var/Inputs/VarData
//   SFI_CasePacker Instance <-> Device 2 (EtherCAT Automation Protocol, EL6601)/Box 97 (Publisher)
//     highest_speed_task Outputs/.RAJ_to_Cartoner <-> RAJ_To_Cartoner_Var/Outputs/VarData
//   SFI_CasePacker Instance <-> Device 2 (EtherCAT Automation Protocol, EL6601)/Box 98 (Subscriber)
//     highest_speed_task Inputs/.Cartoner_to_RAJ <-> Cartoner_To_RAJ_Var/Inputs/VarData
//   SFI_CasePacker Instance <-> Machine Line Connectivity (EtherCAT Automation Protocol)/Box 95 (Publisher)
//     normal_speed_task Outputs/.RAJ_to_Flexlink <-> RAJ_To_Flexlink_Var/Outputs/VarData
//   SFI_CasePacker Instance <-> Machine Line Connectivity (EtherCAT Automation Protocol)/Box 96 (Subscriber)
//     normal_speed_task Inputs/.Flexlink_to_RAJ <-> Flexlink_To_RAJ_Var/Inputs/VarData
//   SFI_CasePacker Instance <-> Machine Line Connectivity (EtherCAT Automation Protocol)/Box 97 (Publisher)
//     highest_speed_task Outputs/.RAJ_to_Cartoner <-> RAJ_To_Cartoner/Outputs/VarData
//   SFI_CasePacker Instance <-> Machine Line Connectivity (EtherCAT Automation Protocol)/Box 98 (Subscriber)
//     highest_speed_task Inputs/.Cartoner_to_RAJ <-> Cartoner_To_RAJ_Var/Inputs/VarData
//   SFI_CasePacker Instance <-> Transfer EtherCAT Master
//     low_speed_task Inputs/csp_main.cabinet_transfer_ethercat_master.field.AmsNetId <-> InfoData/AmsNetId
//     low_speed_task Inputs/csp_main.cabinet_transfer_ethercat_master.field.DevId <-> InfoData/DevId
//     low_speed_task Inputs/csp_main.cabinet_transfer_ethercat_master.field.DevState <-> Inputs/DevState
//   SFI_CasePacker Instance <-> Transfer EtherCAT Master/HMI 6700 (CPXXXX-BK1150)
//     normal_speed_task Inputs/csp_transfer_main_services_pushbuttons.reset_di.field.status <-> Term 6 (CPx9xx-8)/Channel 1/Key 1
//     normal_speed_task Inputs/csp_transfer_main_services_pushbuttons.start_di.field.status <-> Term 6 (CPx9xx-8)/Channel 1/Key 3
//     normal_speed_task Inputs/csp_transfer_main_services_pushbuttons.stop_di.field.status <-> Term 6 (CPx9xx-8)/Channel 1/Key 2
//     normal_speed_task Outputs/csp_transfer_main_services_pushbuttons.reset_lamp_do.field.status <-> Term 6 (CPx9xx-8)/Channel 1/LED 1
//     normal_speed_task Outputs/csp_transfer_main_services_pushbuttons.start_lamp_do.field.status <-> Term 6 (CPx9xx-8)/Channel 1/LED 3
//     normal_speed_task Outputs/csp_transfer_main_services_pushbuttons.stop_lamp_do.field.status <-> Term 6 (CPx9xx-8)/Channel 1/LED 2
//   SFI_CasePacker Instance <-> Transfer EtherCAT Master/IO61600 (EK1100)/IO61600Slot82 (EL7221)
//     low_speed_task Inputs/csp_transfer_infeed_accU_depth.Slot82_drv.process_data_input.status_word <-> DRV Statusword/Statusword
//     low_speed_task Inputs/csp_transfer_infeed_accU_depth.Slot82_drv.process_data_input.torque_actual_value <-> DRV Torque actual value/Torque actual value
//     low_speed_task Inputs/csp_transfer_infeed_accU_depth.axis.hard_increments.value <-> FB Position/Position
//     lowest_speed_task Inputs/csp_transfer_infeed_accU_depth.NC_encoder_val <-> FB Position/Position
//   SFI_CasePacker Instance <-> Transfer EtherCAT Master/IO61600 (EK1100)/IO61600Slot84 (EL7221)
//     low_speed_task Inputs/csp_transfer_infeed_accU_waterfallAdjust.Slot84_drv.process_data_input.status_word <-> DRV Statusword/Statusword
//     low_speed_task Inputs/csp_transfer_infeed_accU_waterfallAdjust.axis.hard_increments.value <-> FB Position/Position
//     lowest_speed_task Inputs/csp_transfer_infeed_accU_waterfallAdjust.NC_encoder_val <-> FB Position/Position
//   SFI_CasePacker Instance <-> Transfer EtherCAT Master/IO61600 (EK1100)/IO61600Slot87 (EL7211)
//     low_speed_task Inputs/csp_transfer_accumulator_accU_depth.Slot87_drv.process_data_input.status_word <-> DRV Statusword/Statusword
//     low_speed_task Inputs/csp_transfer_accumulator_accU_depth.axis.hard_increments.value <-> FB Position/Position
//     lowest_speed_task Inputs/csp_transfer_accumulator_accU_depth.NC_encoder_val <-> FB Position/Position
//   SFI_CasePacker Instance <-> Transfer EtherCAT Master/IO61600 (EK1100)/IO61600Slot89 (EL7211)
//     low_speed_task Inputs/csp_transfer_accumulator_accU_convDepth.Slot89_drv.process_data_input.status_word <-> DRV Statusword/Statusword
//     low_speed_task Inputs/csp_transfer_accumulator_accU_convDepth.axis.hard_increments.value <-> FB Position/Position
//     lowest_speed_task Inputs/csp_transfer_accumulator_accU_convDepth.NC_encoder_val <-> FB Position/Position
//   SFI_CasePacker Instance <-> Transfer EtherCAT Master/IO61600 (EK1100)/IO61600Slot92 (EL7211)
//     low_speed_task Inputs/csp_transfer_accumulator_accU_topRailWidth.Slot92_drv.process_data_input.status_word <-> DRV Statusword/Statusword
//   SFI_CasePacker Instance <-> Transfer EtherCAT Master/IOB40800 (EP1018-0001)
//     highest_speed_task Inputs/csp_transfer_crosspusher_reject.backup_di.field.status <-> Channel 4/Input
//     highest_speed_task Inputs/csp_transfer_crosspusher_reject.present_di.field.status <-> Channel 6/Input
//     highest_speed_task Inputs/csp_transfer_crosspusher_reject.retracted_di.field.status <-> Channel 5/Input
//     highest_speed_task Inputs/csp_transfer_upstacker_backstop.retracted_di.field.status <-> Channel 2/Input
//     highest_speed_task Inputs/csp_transfer_upstacker_sensors.carton_backstop_di.field.status <-> Channel 1/Input
//     highest_speed_task Inputs/csp_transfer_upstacker_sensors.prime_di.field.status <-> Channel 3/Input
//   SFI_CasePacker Instance <-> Transfer EtherCAT Master/IOB40810 (EP2008-0001)
//     highest_speed_task Outputs/csp_transfer_crosspusher_reject.extend_do.field.status <-> Channel 2/Output
//     highest_speed_task Outputs/csp_transfer_upstacker_backstop.extend_do.field.status <-> Channel 1/Output
//   SFI_CasePacker Instance <-> Transfer EtherCAT Master/IOB40820
//     highest_speed_task Inputs/csp_case_loader_pusher.rfid_input_buffer.ByteArr <-> Module 5 (IO-Link Slave)/IO-Link Port3_in/Bitheader 1
//     highest_speed_task Inputs/csp_case_loader_pusher.rfid_input_buffer.ByteArr @bit 72 <-> Module 5 (IO-Link Slave)/IO-Link Port3_in/Bitheader 2
//     highest_speed_task Inputs/csp_case_loader_pusher.rfid_input_buffer.ByteArr @bit {8..64 step 8} <-> Module 5 (IO-Link Slave)/IO-Link Port3_in/Byte {1..8}  (8 links)
//     highest_speed_task Inputs/csp_transfer_crosspusher_sensors.Variable_2bytes <-> Module 4 (IO-Link Slave)/IO-Link Port2/Systemstatus (High-Byte) and Q-Status (Low-Byte)
//     highest_speed_task Inputs/csp_transfer_crosspusher_sensors.output_status_1 <-> Module 4 (IO-Link Slave)/IO-Link Port2/Output Function 1 (QA1)
//     highest_speed_task Outputs/csp_case_loader_pusher.rfid_output_buffer.ByteArr <-> Module 5 (IO-Link Slave)/IO-Link Port3_out/Bitheader 1
//     highest_speed_task Outputs/csp_case_loader_pusher.rfid_output_buffer.ByteArr @bit 72 <-> Module 5 (IO-Link Slave)/IO-Link Port3_out/Bitheader 2
//     highest_speed_task Outputs/csp_case_loader_pusher.rfid_output_buffer.ByteArr @bit {8..64 step 8} <-> Module 5 (IO-Link Slave)/IO-Link Port3_out/Byte {1..8}  (8 links)
//     lowest_speed_task Inputs/csp_transfer_crosspusher_sensors.output_status_2 <-> Module 4 (IO-Link Slave)/IO-Link Port2/Output Function  2 (QA2)
//     normal_speed_task Inputs/csp_transfer_main_ioLink.iol_master_ep6224_IOB40820.CONVERSION_private.process_data_input.AoeNetId <-> InfoData/AoeNetId
//     normal_speed_task Inputs/csp_transfer_main_ioLink.iol_master_ep6224_IOB40820.CONVERSION_private.process_data_input.IOLinkDeviceStateInputs <-> Module 2 (DeviceState Inputs)/DeviceState Inputs/State Ch1
//     normal_speed_task Inputs/csp_transfer_main_ioLink.iol_master_ep6224_IOB40820.CONVERSION_private.process_data_input.IOLinkDeviceStateInputs @bit 8 <-> Module 2 (DeviceState Inputs)/DeviceState Inputs/State Ch2
//     normal_speed_task Inputs/csp_transfer_main_ioLink.iol_master_ep6224_IOB40820.CONVERSION_private.process_data_input.IOLinkDeviceStateInputs @bit 16 <-> Module 2 (DeviceState Inputs)/DeviceState Inputs/State Ch3
//     normal_speed_task Inputs/csp_transfer_main_ioLink.iol_master_ep6224_IOB40820.CONVERSION_private.process_data_input.IOLinkDeviceStateInputs @bit 24 <-> Module 2 (DeviceState Inputs)/DeviceState Inputs/State Ch4
//   SFI_CasePacker Instance <-> Transfer EtherCAT Master/IOB40830 (EP1018-0001)
//     highest_speed_task Inputs/csp_transfer_infeed_reject.bin_full.field.status <-> Channel 7/Input
//     highest_speed_task Inputs/csp_transfer_infeed_reject.bin_present.field.status <-> Channel 6/Input
//     highest_speed_task Inputs/csp_transfer_infeed_reject.os_chute_backup.field.status <-> Channel 8/Input
//     low_speed_task Inputs/csp_transfer_infeed_accumulation_level_low.di.field.status <-> Channel 2/Input
//     low_speed_task Inputs/csp_transfer_infeed_accumulation_level_max.di.field.status <-> Channel 3/Input
//     low_speed_task Inputs/csp_transfer_infeed_accumulation_level_min.di.field.status <-> Channel 1/Input
//     low_speed_task Inputs/csp_transfer_infeed_accumulation_level_normal.di.field.status <-> Channel 5/Input
//     low_speed_task Inputs/csp_transfer_infeed_metering_jam.jam_di.field.status <-> Channel 4/Input
//   SFI_CasePacker Instance <-> Transfer EtherCAT Master/IOB40900 (EP2318-0001)
//     highest_speed_task Inputs/csp_transfer_infeed_barcode_reader.barcode_trigger_di_downstream.field.status <-> Channel 4/Input
//     highest_speed_task Inputs/csp_transfer_infeed_barcode_reader.barcode_trigger_di_upstream.field.status <-> Channel 3/Input
//     highest_speed_task Inputs/csp_transfer_infeed_clamp.ls_retracted_di.field.status <-> Channel 2/Input
//     highest_speed_task Inputs/csp_transfer_infeed_clamp.os_retracted_di.field.status <-> Channel 1/Input
//     highest_speed_task Outputs/csp_transfer_infeed_clamp.extend_do.field.status <-> Channel 5/Output
//   SFI_CasePacker Instance <-> Transfer EtherCAT Master/IOB40909
//     highest_speed_task Inputs/csp_transfer_infeed_reject_highLoad.Variable_2bytes <-> Module 4 (IO-Link Slave)/IO-Link Port2/Systemstatus (High-Byte) and Q-Status (Low-Byte)
//     highest_speed_task Inputs/csp_transfer_infeed_reject_highLoad.output_status_1 <-> Module 4 (IO-Link Slave)/IO-Link Port2/Output Function 1 (QA1)
//     lowest_speed_task Inputs/csp_transfer_infeed_reject_highLoad.output_status_2 <-> Module 4 (IO-Link Slave)/IO-Link Port2/Output Function  2 (QA2)
//     normal_speed_task Inputs/csp_transfer_main_ioLink.iol_master_ep6224_IOB40909.CONVERSION_private.process_data_input.AoeNetId <-> InfoData/AoeNetId
//     normal_speed_task Inputs/csp_transfer_main_ioLink.iol_master_ep6224_IOB40909.CONVERSION_private.process_data_input.IOLinkDeviceStateInputs <-> Module 2 (DeviceState Inputs)/DeviceState Inputs/State Ch1
//     normal_speed_task Inputs/csp_transfer_main_ioLink.iol_master_ep6224_IOB40909.CONVERSION_private.process_data_input.IOLinkDeviceStateInputs @bit 8 <-> Module 2 (DeviceState Inputs)/DeviceState Inputs/State Ch2
//     normal_speed_task Inputs/csp_transfer_main_ioLink.iol_master_ep6224_IOB40909.CONVERSION_private.process_data_input.IOLinkDeviceStateInputs @bit 16 <-> Module 2 (DeviceState Inputs)/DeviceState Inputs/State Ch3
//     normal_speed_task Inputs/csp_transfer_main_ioLink.iol_master_ep6224_IOB40909.CONVERSION_private.process_data_input.IOLinkDeviceStateInputs @bit 24 <-> Module 2 (DeviceState Inputs)/DeviceState Inputs/State Ch4
//   SFI_CasePacker Instance <-> Transfer EtherCAT Master/SD41100
//     highest_speed_task Inputs/csp_transfer_main_drives.SD41100_drv.channel_a.process_data_input.dc_bus_power <-> AT 1/DC bus power
//     highest_speed_task Inputs/csp_transfer_main_drives.SD41100_drv.channel_a.process_data_input.dc_bus_voltage <-> AT 1/DC bus voltage
//     highest_speed_task Inputs/csp_transfer_main_drives.SD41100_drv.channel_a.process_data_input.motor_temperature <-> AT 1/Motor temperature
//     highest_speed_task Inputs/csp_transfer_main_drives.SD41100_drv.channel_b.process_data_input.dc_bus_power <-> AT 2/DC bus power
//     highest_speed_task Inputs/csp_transfer_main_drives.SD41100_drv.channel_b.process_data_input.dc_bus_voltage <-> AT 2/DC bus voltage
//     highest_speed_task Inputs/csp_transfer_main_drives.SD41100_drv.channel_b.process_data_input.motor_temperature <-> AT 2/Motor temperature
//     normal_speed_task Inputs/csp_transfer_main_drives.SD41100_drv.channel_a.process_data_input.actual_absolute_current <-> AT 1/Torque-generating current, actual value
//     normal_speed_task Inputs/csp_transfer_main_drives.SD41100_drv.channel_a.process_data_input.dc_bus_ready <-> AT 1/Device control: Status word[15]
//     normal_speed_task Inputs/csp_transfer_main_drives.SD41100_drv.channel_a.process_data_input.status_parametrization_level <-> AT 1/Status parametrization level
//     normal_speed_task Inputs/csp_transfer_main_drives.SD41100_drv.channel_a.process_data_input.warning_active <-> AT 1/Device control: Status word[2]
//     normal_speed_task Inputs/csp_transfer_main_drives.SD41100_drv.channel_b.process_data_input.actual_absolute_current <-> AT 2/Torque-generating current, actual value
//     normal_speed_task Inputs/csp_transfer_main_drives.SD41100_drv.channel_b.process_data_input.dc_bus_ready <-> AT 2/Device control: Status word[15]
//     normal_speed_task Inputs/csp_transfer_main_drives.SD41100_drv.channel_b.process_data_input.status_parametrization_level <-> AT 2/Status parametrization level
//     normal_speed_task Inputs/csp_transfer_main_drives.SD41100_drv.channel_b.process_data_input.warning_active <-> AT 2/Device control: Status word[2]
//   SFI_CasePacker Instance <-> Transfer EtherCAT Master/SD41200
//     normal_speed_task Inputs/csp_transfer_main_drives.SD41200_drv.channel_a.process_data_input.actual_absolute_current <-> AT 1/Torque-generating current, actual value
//     normal_speed_task Inputs/csp_transfer_main_drives.SD41200_drv.channel_a.process_data_input.dc_bus_power <-> AT 1/DC bus power
//     normal_speed_task Inputs/csp_transfer_main_drives.SD41200_drv.channel_a.process_data_input.dc_bus_ready <-> AT 1/Device control: Status word[15]
//     normal_speed_task Inputs/csp_transfer_main_drives.SD41200_drv.channel_a.process_data_input.dc_bus_voltage <-> AT 1/DC bus voltage
//     normal_speed_task Inputs/csp_transfer_main_drives.SD41200_drv.channel_a.process_data_input.motor_temperature <-> AT 1/Motor temperature
//     normal_speed_task Inputs/csp_transfer_main_drives.SD41200_drv.channel_a.process_data_input.status_parametrization_level <-> AT 1/Status parametrization level
//     normal_speed_task Inputs/csp_transfer_main_drives.SD41200_drv.channel_a.process_data_input.warning_active <-> AT 1/Device control: Status word[2]
//     normal_speed_task Inputs/csp_transfer_main_drives.SD41200_drv.channel_b.process_data_input.actual_absolute_current <-> AT 2/Torque-generating current, actual value
//     normal_speed_task Inputs/csp_transfer_main_drives.SD41200_drv.channel_b.process_data_input.dc_bus_power <-> AT 2/DC bus power
//     normal_speed_task Inputs/csp_transfer_main_drives.SD41200_drv.channel_b.process_data_input.dc_bus_ready <-> AT 2/Device control: Status word[15]
//     normal_speed_task Inputs/csp_transfer_main_drives.SD41200_drv.channel_b.process_data_input.dc_bus_voltage <-> AT 2/DC bus voltage
//     normal_speed_task Inputs/csp_transfer_main_drives.SD41200_drv.channel_b.process_data_input.motor_temperature <-> AT 2/Motor temperature
//     normal_speed_task Inputs/csp_transfer_main_drives.SD41200_drv.channel_b.process_data_input.status_parametrization_level <-> AT 2/Status parametrization level
//     normal_speed_task Inputs/csp_transfer_main_drives.SD41200_drv.channel_b.process_data_input.warning_active <-> AT 2/Device control: Status word[2]
//   SFI_CasePacker Instance <-> Transfer EtherCAT Master/SD41300
//     highest_speed_task Inputs/csp_transfer_main_drives.SD41300_drv.channel_a.process_data_input.dc_bus_power <-> AT 1/DC bus power
//     highest_speed_task Inputs/csp_transfer_main_drives.SD41300_drv.channel_a.process_data_input.dc_bus_voltage <-> AT 1/DC bus voltage
//     highest_speed_task Inputs/csp_transfer_main_drives.SD41300_drv.channel_a.process_data_input.motor_temperature <-> AT 1/Motor temperature
//     highest_speed_task Inputs/csp_transfer_main_drives.SD41300_drv.channel_b.process_data_input.dc_bus_power <-> AT 2/DC bus power
//     highest_speed_task Inputs/csp_transfer_main_drives.SD41300_drv.channel_b.process_data_input.dc_bus_voltage <-> AT 2/DC bus voltage
//     highest_speed_task Inputs/csp_transfer_main_drives.SD41300_drv.channel_b.process_data_input.motor_temperature <-> AT 2/Motor temperature
//     normal_speed_task Inputs/csp_transfer_main_drives.SD41300_drv.channel_a.process_data_input.actual_absolute_current <-> AT 1/Torque-generating current, actual value
//     normal_speed_task Inputs/csp_transfer_main_drives.SD41300_drv.channel_a.process_data_input.dc_bus_ready <-> AT 1/Device control: Status word[15]
//     normal_speed_task Inputs/csp_transfer_main_drives.SD41300_drv.channel_a.process_data_input.status_parametrization_level <-> AT 1/Status parametrization level
//     normal_speed_task Inputs/csp_transfer_main_drives.SD41300_drv.channel_a.process_data_input.warning_active <-> AT 1/Device control: Status word[2]
//     normal_speed_task Inputs/csp_transfer_main_drives.SD41300_drv.channel_b.process_data_input.actual_absolute_current <-> AT 2/Torque-generating current, actual value
//     normal_speed_task Inputs/csp_transfer_main_drives.SD41300_drv.channel_b.process_data_input.dc_bus_ready <-> AT 2/Device control: Status word[15]
//     normal_speed_task Inputs/csp_transfer_main_drives.SD41300_drv.channel_b.process_data_input.status_parametrization_level <-> AT 2/Status parametrization level
//     normal_speed_task Inputs/csp_transfer_main_drives.SD41300_drv.channel_b.process_data_input.warning_active <-> AT 2/Device control: Status word[2]
//   SFI_CasePacker Instance <-> Transfer EtherCAT Master/SD41400
//     highest_speed_task Inputs/csp_transfer_main_drives.SD41400_drv.channel_a.process_data_input.dc_bus_power <-> AT 1/DC bus power
//     highest_speed_task Inputs/csp_transfer_main_drives.SD41400_drv.channel_a.process_data_input.dc_bus_voltage <-> AT 1/DC bus voltage
//     highest_speed_task Inputs/csp_transfer_main_drives.SD41400_drv.channel_a.process_data_input.motor_temperature <-> AT 1/Motor temperature
//     highest_speed_task Inputs/csp_transfer_main_drives.SD41400_drv.channel_b.process_data_input.dc_bus_power <-> AT 2/DC bus power
//     highest_speed_task Inputs/csp_transfer_main_drives.SD41400_drv.channel_b.process_data_input.dc_bus_voltage <-> AT 2/DC bus voltage
//     highest_speed_task Inputs/csp_transfer_main_drives.SD41400_drv.channel_b.process_data_input.motor_temperature <-> AT 2/Motor temperature
//     normal_speed_task Inputs/csp_transfer_main_drives.SD41400_drv.channel_a.process_data_input.actual_absolute_current <-> AT 1/Torque-generating current, actual value
//     normal_speed_task Inputs/csp_transfer_main_drives.SD41400_drv.channel_a.process_data_input.dc_bus_ready <-> AT 1/Device control: Status word[15]
//     normal_speed_task Inputs/csp_transfer_main_drives.SD41400_drv.channel_a.process_data_input.status_parametrization_level <-> AT 1/Status parametrization level
//     normal_speed_task Inputs/csp_transfer_main_drives.SD41400_drv.channel_a.process_data_input.warning_active <-> AT 1/Device control: Status word[2]
//     normal_speed_task Inputs/csp_transfer_main_drives.SD41400_drv.channel_b.process_data_input.actual_absolute_current <-> AT 2/Torque-generating current, actual value
//     normal_speed_task Inputs/csp_transfer_main_drives.SD41400_drv.channel_b.process_data_input.dc_bus_ready <-> AT 2/Device control: Status word[15]
//     normal_speed_task Inputs/csp_transfer_main_drives.SD41400_drv.channel_b.process_data_input.status_parametrization_level <-> AT 2/Status parametrization level
//     normal_speed_task Inputs/csp_transfer_main_drives.SD41400_drv.channel_b.process_data_input.warning_active <-> AT 2/Device control: Status word[2]
//   SFI_CasePacker Instance <-> Transfer EtherCAT Master/SD41500
//     highest_speed_task Inputs/csp_transfer_main_drives.SD41500_drv.channel_a.process_data_input.dc_bus_power <-> AT 1/DC bus power
//     highest_speed_task Inputs/csp_transfer_main_drives.SD41500_drv.channel_a.process_data_input.dc_bus_voltage <-> AT 1/DC bus voltage
//     highest_speed_task Inputs/csp_transfer_main_drives.SD41500_drv.channel_a.process_data_input.motor_temperature <-> AT 1/Motor temperature
//     highest_speed_task Inputs/csp_transfer_main_drives.SD41500_drv.channel_b.process_data_input.dc_bus_power <-> AT 2/DC bus power
//     highest_speed_task Inputs/csp_transfer_main_drives.SD41500_drv.channel_b.process_data_input.dc_bus_voltage <-> AT 2/DC bus voltage
//     highest_speed_task Inputs/csp_transfer_main_drives.SD41500_drv.channel_b.process_data_input.motor_temperature <-> AT 2/Motor temperature
//     normal_speed_task Inputs/csp_transfer_main_drives.SD41500_drv.channel_a.process_data_input.actual_absolute_current <-> AT 1/Torque-generating current, actual value
//     normal_speed_task Inputs/csp_transfer_main_drives.SD41500_drv.channel_a.process_data_input.dc_bus_ready <-> AT 1/Device control: Status word[15]
//     normal_speed_task Inputs/csp_transfer_main_drives.SD41500_drv.channel_a.process_data_input.status_parametrization_level <-> AT 1/Status parametrization level
//     normal_speed_task Inputs/csp_transfer_main_drives.SD41500_drv.channel_a.process_data_input.warning_active <-> AT 1/Device control: Status word[2]
//     normal_speed_task Inputs/csp_transfer_main_drives.SD41500_drv.channel_b.process_data_input.actual_absolute_current <-> AT 2/Torque-generating current, actual value
//     normal_speed_task Inputs/csp_transfer_main_drives.SD41500_drv.channel_b.process_data_input.dc_bus_ready <-> AT 2/Device control: Status word[15]
//     normal_speed_task Inputs/csp_transfer_main_drives.SD41500_drv.channel_b.process_data_input.status_parametrization_level <-> AT 2/Status parametrization level
//     normal_speed_task Inputs/csp_transfer_main_drives.SD41500_drv.channel_b.process_data_input.warning_active <-> AT 2/Device control: Status word[2]
//   SFI_CasePacker Instance <-> Transfer EtherCAT Master/SD41600
//     normal_speed_task Inputs/csp_transfer_main_drives.SD41600_drv.channel_a.process_data_input.actual_absolute_current <-> AT 1/Torque-generating current, actual value
//     normal_speed_task Inputs/csp_transfer_main_drives.SD41600_drv.channel_a.process_data_input.dc_bus_power <-> AT 1/DC bus power
//     normal_speed_task Inputs/csp_transfer_main_drives.SD41600_drv.channel_a.process_data_input.dc_bus_ready <-> AT 1/Device control: Status word[15]
//     normal_speed_task Inputs/csp_transfer_main_drives.SD41600_drv.channel_a.process_data_input.dc_bus_voltage <-> AT 1/DC bus voltage
//     normal_speed_task Inputs/csp_transfer_main_drives.SD41600_drv.channel_a.process_data_input.motor_temperature <-> AT 1/Motor temperature
//     normal_speed_task Inputs/csp_transfer_main_drives.SD41600_drv.channel_a.process_data_input.status_parametrization_level <-> AT 1/Status parametrization level
//     normal_speed_task Inputs/csp_transfer_main_drives.SD41600_drv.channel_a.process_data_input.warning_active <-> AT 1/Device control: Status word[2]
//     normal_speed_task Inputs/csp_transfer_main_drives.SD41600_drv.channel_b.process_data_input.actual_absolute_current <-> AT 2/Torque-generating current, actual value
//     normal_speed_task Inputs/csp_transfer_main_drives.SD41600_drv.channel_b.process_data_input.dc_bus_power <-> AT 2/DC bus power
//     normal_speed_task Inputs/csp_transfer_main_drives.SD41600_drv.channel_b.process_data_input.dc_bus_ready <-> AT 2/Device control: Status word[15]
//     normal_speed_task Inputs/csp_transfer_main_drives.SD41600_drv.channel_b.process_data_input.dc_bus_voltage <-> AT 2/DC bus voltage
//     normal_speed_task Inputs/csp_transfer_main_drives.SD41600_drv.channel_b.process_data_input.motor_temperature <-> AT 2/Motor temperature
//     normal_speed_task Inputs/csp_transfer_main_drives.SD41600_drv.channel_b.process_data_input.status_parametrization_level <-> AT 2/Status parametrization level
//     normal_speed_task Inputs/csp_transfer_main_drives.SD41600_drv.channel_b.process_data_input.warning_active <-> AT 2/Device control: Status word[2]
//   SFI_CasePacker Instance <-> Transfer EtherCAT Master/SD41700
//     normal_speed_task Inputs/csp_transfer_main_drives.SD41700_drv.channel_a.process_data_input.actual_absolute_current <-> AT 1/Torque-generating current, actual value
//     normal_speed_task Inputs/csp_transfer_main_drives.SD41700_drv.channel_a.process_data_input.dc_bus_power <-> AT 1/DC bus power
//     normal_speed_task Inputs/csp_transfer_main_drives.SD41700_drv.channel_a.process_data_input.dc_bus_ready <-> AT 1/Device control: Status word[15]
//     normal_speed_task Inputs/csp_transfer_main_drives.SD41700_drv.channel_a.process_data_input.dc_bus_voltage <-> AT 1/DC bus voltage
//     normal_speed_task Inputs/csp_transfer_main_drives.SD41700_drv.channel_a.process_data_input.motor_temperature <-> AT 1/Motor temperature
